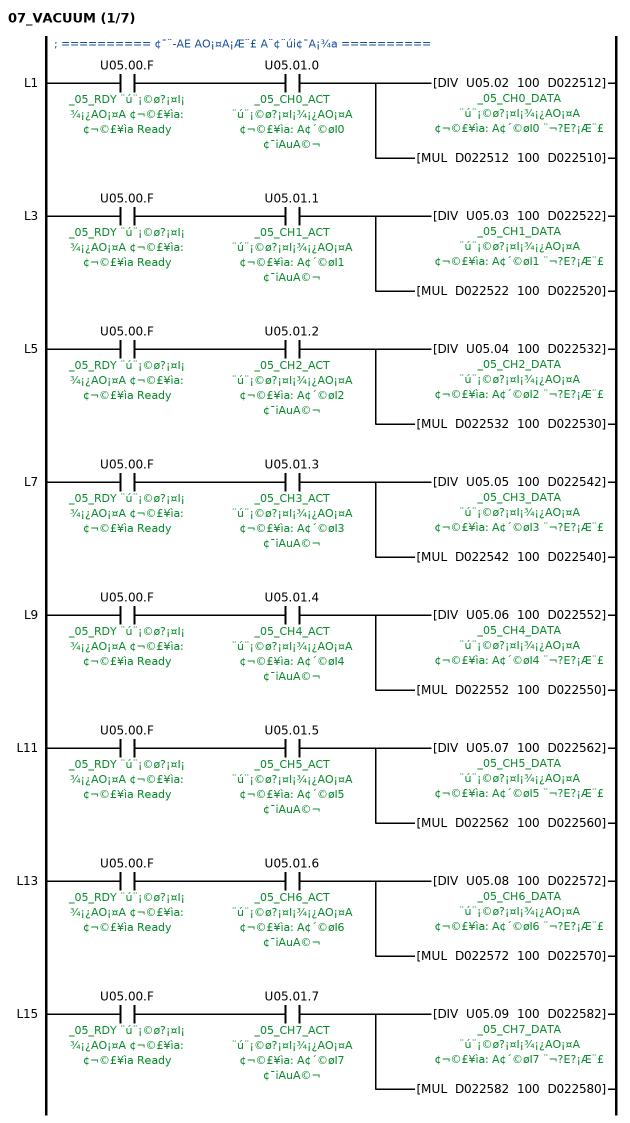
[picture p48: 07_VACUUM rungs L1-L15]
// ========== ¢¯¨­AE AO¡¤A¡Æ¨£ A¨¢¨úi¢¯A¡¾a ==========
; L1
LOAD      U05.00.F	// _05_RDY ¨ú¨¡©ø?¡¤I¡¾¡¿AO¡¤A ¢¬©£¥ìa: ¢¬©£¥ìa Ready
AND       U05.01.0	// _05_CH0_ACT ¨ú¨¡©ø?¡¤I¡¾¡¿AO¡¤A ¢¬©£¥ìa: A¢´©øI0 ¢¯iAuA©¬
DIV       U05.02 100 D022512	// _05_CH0_DATA ¨ú¨¡©ø?¡¤I¡¾¡¿AO¡¤A ¢¬©£¥ìa: A¢´©øI0 ¨¬?E?¡Æ¨£
MUL       D022512 100 D022510
; L3
LOAD      U05.00.F	// _05_RDY ¨ú¨¡©ø?¡¤I¡¾¡¿AO¡¤A ¢¬©£¥ìa: ¢¬©£¥ìa Ready
AND       U05.01.1	// _05_CH1_ACT ¨ú¨¡©ø?¡¤I¡¾¡¿AO¡¤A ¢¬©£¥ìa: A¢´©øI1 ¢¯iAuA©¬
DIV       U05.03 100 D022522	// _05_CH1_DATA ¨ú¨¡©ø?¡¤I¡¾¡¿AO¡¤A ¢¬©£¥ìa: A¢´©øI1 ¨¬?E?¡Æ¨£
MUL       D022522 100 D022520
; L5
LOAD      U05.00.F	// _05_RDY ¨ú¨¡©ø?¡¤I¡¾¡¿AO¡¤A ¢¬©£¥ìa: ¢¬©£¥ìa Ready
AND       U05.01.2	// _05_CH2_ACT ¨ú¨¡©ø?¡¤I¡¾¡¿AO¡¤A ¢¬©£¥ìa: A¢´©øI2 ¢¯iAuA©¬
DIV       U05.04 100 D022532	// _05_CH2_DATA ¨ú¨¡©ø?¡¤I¡¾¡¿AO¡¤A ¢¬©£¥ìa: A¢´©øI2 ¨¬?E?¡Æ¨£
MUL       D022532 100 D022530
; L7
LOAD      U05.00.F	// _05_RDY ¨ú¨¡©ø?¡¤I¡¾¡¿AO¡¤A ¢¬©£¥ìa: ¢¬©£¥ìa Ready
AND       U05.01.3	// _05_CH3_ACT ¨ú¨¡©ø?¡¤I¡¾¡¿AO¡¤A ¢¬©£¥ìa: A¢´©øI3 ¢¯iAuA©¬
DIV       U05.05 100 D022542	// _05_CH3_DATA ¨ú¨¡©ø?¡¤I¡¾¡¿AO¡¤A ¢¬©£¥ìa: A¢´©øI3 ¨¬?E?¡Æ¨£
MUL       D022542 100 D022540
; L9
LOAD      U05.00.F	// _05_RDY ¨ú¨¡©ø?¡¤I¡¾¡¿AO¡¤A ¢¬©£¥ìa: ¢¬©£¥ìa Ready
AND       U05.01.4	// _05_CH4_ACT ¨ú¨¡©ø?¡¤I¡¾¡¿AO¡¤A ¢¬©£¥ìa: A¢´©øI4 ¢¯iAuA©¬
DIV       U05.06 100 D022552	// _05_CH4_DATA ¨ú¨¡©ø?¡¤I¡¾¡¿AO¡¤A ¢¬©£¥ìa: A¢´©øI4 ¨¬?E?¡Æ¨£
MUL       D022552 100 D022550
; L11
LOAD      U05.00.F	// _05_RDY ¨ú¨¡©ø?¡¤I¡¾¡¿AO¡¤A ¢¬©£¥ìa: ¢¬©£¥ìa Ready
AND       U05.01.5	// _05_CH5_ACT ¨ú¨¡©ø?¡¤I¡¾¡¿AO¡¤A ¢¬©£¥ìa: A¢´©øI5 ¢¯iAuA©¬
DIV       U05.07 100 D022562	// _05_CH5_DATA ¨ú¨¡©ø?¡¤I¡¾¡¿AO¡¤A ¢¬©£¥ìa: A¢´©øI5 ¨¬?E?¡Æ¨£
MUL       D022562 100 D022560
; L13
LOAD      U05.00.F	// _05_RDY ¨ú¨¡©ø?¡¤I¡¾¡¿AO¡¤A ¢¬©£¥ìa: ¢¬©£¥ìa Ready
AND       U05.01.6	// _05_CH6_ACT ¨ú¨¡©ø?¡¤I¡¾¡¿AO¡¤A ¢¬©£¥ìa: A¢´©øI6 ¢¯iAuA©¬
DIV       U05.08 100 D022572	// _05_CH6_DATA ¨ú¨¡©ø?¡¤I¡¾¡¿AO¡¤A ¢¬©£¥ìa: A¢´©øI6 ¨¬?E?¡Æ¨£
MUL       D022572 100 D022570
; L15
LOAD      U05.00.F	// _05_RDY ¨ú¨¡©ø?¡¤I¡¾¡¿AO¡¤A ¢¬©£¥ìa: ¢¬©£¥ìa Ready
AND       U05.01.7	// _05_CH7_ACT ¨ú¨¡©ø?¡¤I¡¾¡¿AO¡¤A ¢¬©£¥ìa: A¢´©øI7 ¢¯iAuA©¬
DIV       U05.09 100 D022582	// _05_CH7_DATA ¨ú¨¡©ø?¡¤I¡¾¡¿AO¡¤A ¢¬©£¥ìa: A¢´©øI7 ¨¬?E?¡Æ¨£
MUL       D022582 100 D022580

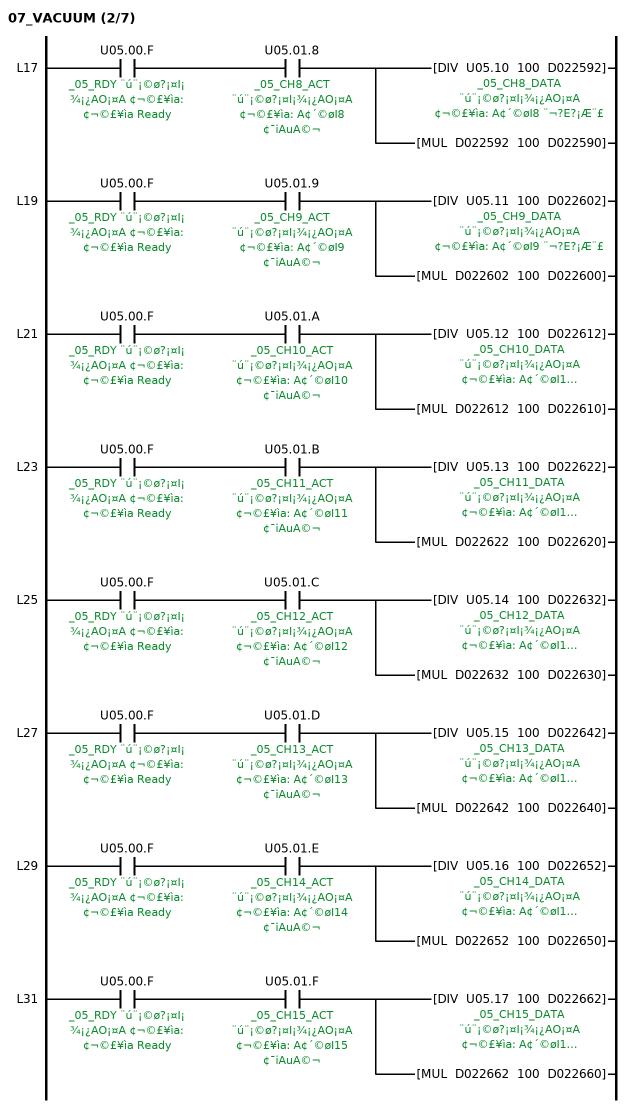
; L17
LOAD      U05.00.F	// _05_RDY ¨ú¨¡©ø?¡¤I¡¾¡¿AO¡¤A ¢¬©£¥ìa: ¢¬©£¥ìa Ready
AND       U05.01.8	// _05_CH8_ACT ¨ú¨¡©ø?¡¤I¡¾¡¿AO¡¤A ¢¬©£¥ìa: A¢´©øI8 ¢¯iAuA©¬
DIV       U05.10 100 D022592	// _05_CH8_DATA ¨ú¨¡©ø?¡¤I¡¾¡¿AO¡¤A ¢¬©£¥ìa: A¢´©øI8 ¨¬?E?¡Æ¨£
MUL       D022592 100 D022590
; L19
LOAD      U05.00.F	// _05_RDY ¨ú¨¡©ø?¡¤I¡¾¡¿AO¡¤A ¢¬©£¥ìa: ¢¬©£¥ìa Ready
AND       U05.01.9	// _05_CH9_ACT ¨ú¨¡©ø?¡¤I¡¾¡¿AO¡¤A ¢¬©£¥ìa: A¢´©øI9 ¢¯iAuA©¬
DIV       U05.11 100 D022602	// _05_CH9_DATA ¨ú¨¡©ø?¡¤I¡¾¡¿AO¡¤A ¢¬©£¥ìa: A¢´©øI9 ¨¬?E?¡Æ¨£
MUL       D022602 100 D022600
; L21
LOAD      U05.00.F	// _05_RDY ¨ú¨¡©ø?¡¤I¡¾¡¿AO¡¤A ¢¬©£¥ìa: ¢¬©£¥ìa Ready
AND       U05.01.A	// _05_CH10_ACT ¨ú¨¡©ø?¡¤I¡¾¡¿AO¡¤A ¢¬©£¥ìa: A¢´©øI10 ¢¯iAuA©¬
DIV       U05.12 100 D022612	// _05_CH10_DATA ¨ú¨¡©ø?¡¤I¡¾¡¿AO¡¤A ¢¬©£¥ìa: A¢´©øI10 ¨¬?E?¡Æ¨£
MUL       D022612 100 D022610
; L23
LOAD      U05.00.F	// _05_RDY ¨ú¨¡©ø?¡¤I¡¾¡¿AO¡¤A ¢¬©£¥ìa: ¢¬©£¥ìa Ready
AND       U05.01.B	// _05_CH11_ACT ¨ú¨¡©ø?¡¤I¡¾¡¿AO¡¤A ¢¬©£¥ìa: A¢´©øI11 ¢¯iAuA©¬
DIV       U05.13 100 D022622	// _05_CH11_DATA ¨ú¨¡©ø?¡¤I¡¾¡¿AO¡¤A ¢¬©£¥ìa: A¢´©øI11 ¨¬?E?¡Æ¨£
MUL       D022622 100 D022620
; L25
LOAD      U05.00.F	// _05_RDY ¨ú¨¡©ø?¡¤I¡¾¡¿AO¡¤A ¢¬©£¥ìa: ¢¬©£¥ìa Ready
AND       U05.01.C	// _05_CH12_ACT ¨ú¨¡©ø?¡¤I¡¾¡¿AO¡¤A ¢¬©£¥ìa: A¢´©øI12 ¢¯iAuA©¬
DIV       U05.14 100 D022632	// _05_CH12_DATA ¨ú¨¡©ø?¡¤I¡¾¡¿AO¡¤A ¢¬©£¥ìa: A¢´©øI12 ¨¬?E?¡Æ¨£
MUL       D022632 100 D022630
; L27
LOAD      U05.00.F	// _05_RDY ¨ú¨¡©ø?¡¤I¡¾¡¿AO¡¤A ¢¬©£¥ìa: ¢¬©£¥ìa Ready
AND       U05.01.D	// _05_CH13_ACT ¨ú¨¡©ø?¡¤I¡¾¡¿AO¡¤A ¢¬©£¥ìa: A¢´©øI13 ¢¯iAuA©¬
DIV       U05.15 100 D022642	// _05_CH13_DATA ¨ú¨¡©ø?¡¤I¡¾¡¿AO¡¤A ¢¬©£¥ìa: A¢´©øI13 ¨¬?E?¡Æ¨£
MUL       D022642 100 D022640
; L29
LOAD      U05.00.F	// _05_RDY ¨ú¨¡©ø?¡¤I¡¾¡¿AO¡¤A ¢¬©£¥ìa: ¢¬©£¥ìa Ready
AND       U05.01.E	// _05_CH14_ACT ¨ú¨¡©ø?¡¤I¡¾¡¿AO¡¤A ¢¬©£¥ìa: A¢´©øI14 ¢¯iAuA©¬
DIV       U05.16 100 D022652	// _05_CH14_DATA ¨ú¨¡©ø?¡¤I¡¾¡¿AO¡¤A ¢¬©£¥ìa: A¢´©øI14 ¨¬?E?¡Æ¨£
MUL       D022652 100 D022650
; L31
LOAD      U05.00.F	// _05_RDY ¨ú¨¡©ø?¡¤I¡¾¡¿AO¡¤A ¢¬©£¥ìa: ¢¬©£¥ìa Ready
AND       U05.01.F	// _05_CH15_ACT ¨ú¨¡©ø?¡¤I¡¾¡¿AO¡¤A ¢¬©£¥ìa: A¢´©øI15 ¢¯iAuA©¬
DIV       U05.17 100 D022662	// _05_CH15_DATA ¨ú¨¡©ø?¡¤I¡¾¡¿AO¡¤A ¢¬©£¥ìa: A¢´©øI15 ¨¬?E?¡Æ¨£
MUL       D022662 100 D022660

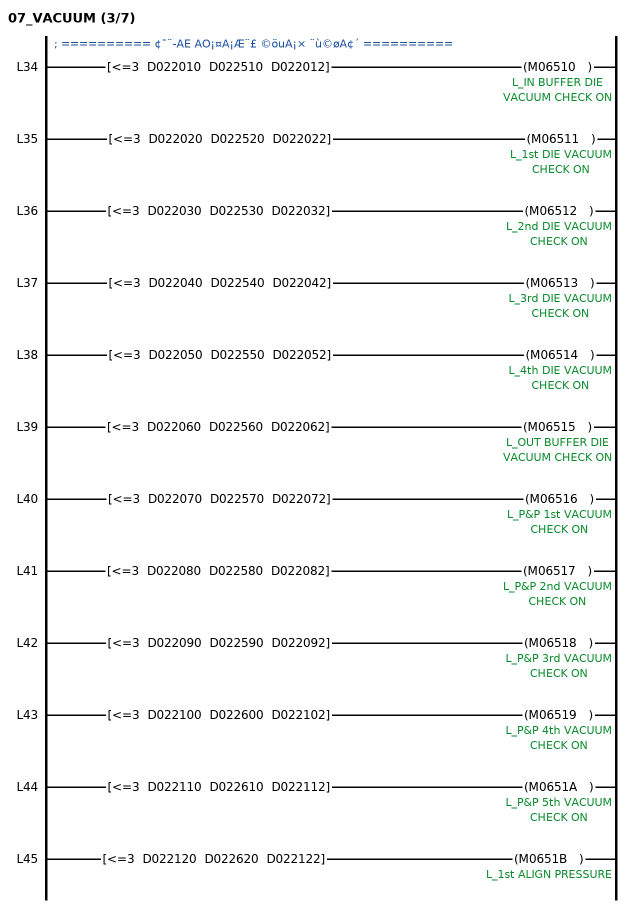
// ========== ¢¯¨­AE AO¡¤A¡Æ¨£ ©öuA¡× ¨ù©øA¢´ ==========
; L34
LOAD<=3   D022010 D022510 D022012
OUT       M06510	// L_IN BUFFER DIE VACUUM CHECK ON
; L35
LOAD<=3   D022020 D022520 D022022
OUT       M06511	// L_1st DIE VACUUM CHECK ON
; L36
LOAD<=3   D022030 D022530 D022032
OUT       M06512	// L_2nd DIE VACUUM CHECK ON
; L37
LOAD<=3   D022040 D022540 D022042
OUT       M06513	// L_3rd DIE VACUUM CHECK ON
; L38
LOAD<=3   D022050 D022550 D022052
OUT       M06514	// L_4th DIE VACUUM CHECK ON
; L39
LOAD<=3   D022060 D022560 D022062
OUT       M06515	// L_OUT BUFFER DIE VACUUM CHECK ON
; L40
LOAD<=3   D022070 D022570 D022072
OUT       M06516	// L_P&P 1st VACUUM CHECK ON
; L41
LOAD<=3   D022080 D022580 D022082
OUT       M06517	// L_P&P 2nd VACUUM CHECK ON
; L42
LOAD<=3   D022090 D022590 D022092
OUT       M06518	// L_P&P 3rd VACUUM CHECK ON
; L43
LOAD<=3   D022100 D022600 D022102
OUT       M06519	// L_P&P 4th VACUUM CHECK ON
; L44
LOAD<=3   D022110 D022610 D022112
OUT       M0651A	// L_P&P 5th VACUUM CHECK ON
; L45
LOAD<=3   D022120 D022620 D022122
OUT       M0651B	// L_1st ALIGN PRESSURE

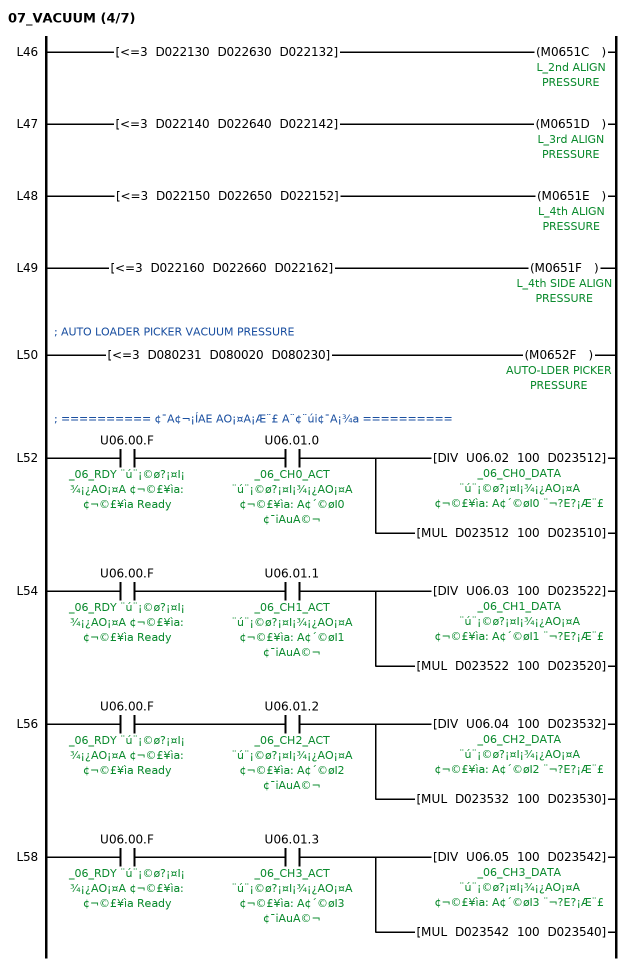
; L46
LOAD<=3   D022130 D022630 D022132
OUT       M0651C	// L_2nd ALIGN PRESSURE
; L47
LOAD<=3   D022140 D022640 D022142
OUT       M0651D	// L_3rd ALIGN PRESSURE
; L48
LOAD<=3   D022150 D022650 D022152
OUT       M0651E	// L_4th ALIGN PRESSURE
; L49
LOAD<=3   D022160 D022660 D022162
OUT       M0651F	// L_4th SIDE ALIGN PRESSURE
; L50
LOAD<=3   D080231 D080020 D080230
OUT       M0652F	// AUTO-LDER PICKER PRESSURE
// output comment: AUTO LOADER PICKER VACUUM PRESSURE
// ========== ¢¯A¢¬¡ÍAE AO¡¤A¡Æ¨£ A¨¢¨úi¢¯A¡¾a ==========
; L52
LOAD      U06.00.F	// _06_RDY ¨ú¨¡©ø?¡¤I¡¾¡¿AO¡¤A ¢¬©£¥ìa: ¢¬©£¥ìa Ready
AND       U06.01.0	// _06_CH0_ACT ¨ú¨¡©ø?¡¤I¡¾¡¿AO¡¤A ¢¬©£¥ìa: A¢´©øI0 ¢¯iAuA©¬
DIV       U06.02 100 D023512	// _06_CH0_DATA ¨ú¨¡©ø?¡¤I¡¾¡¿AO¡¤A ¢¬©£¥ìa: A¢´©øI0 ¨¬?E?¡Æ¨£
MUL       D023512 100 D023510
; L54
LOAD      U06.00.F	// _06_RDY ¨ú¨¡©ø?¡¤I¡¾¡¿AO¡¤A ¢¬©£¥ìa: ¢¬©£¥ìa Ready
AND       U06.01.1	// _06_CH1_ACT ¨ú¨¡©ø?¡¤I¡¾¡¿AO¡¤A ¢¬©£¥ìa: A¢´©øI1 ¢¯iAuA©¬
DIV       U06.03 100 D023522	// _06_CH1_DATA ¨ú¨¡©ø?¡¤I¡¾¡¿AO¡¤A ¢¬©£¥ìa: A¢´©øI1 ¨¬?E?¡Æ¨£
MUL       D023522 100 D023520
; L56
LOAD      U06.00.F	// _06_RDY ¨ú¨¡©ø?¡¤I¡¾¡¿AO¡¤A ¢¬©£¥ìa: ¢¬©£¥ìa Ready
AND       U06.01.2	// _06_CH2_ACT ¨ú¨¡©ø?¡¤I¡¾¡¿AO¡¤A ¢¬©£¥ìa: A¢´©øI2 ¢¯iAuA©¬
DIV       U06.04 100 D023532	// _06_CH2_DATA ¨ú¨¡©ø?¡¤I¡¾¡¿AO¡¤A ¢¬©£¥ìa: A¢´©øI2 ¨¬?E?¡Æ¨£
MUL       D023532 100 D023530
; L58
LOAD      U06.00.F	// _06_RDY ¨ú¨¡©ø?¡¤I¡¾¡¿AO¡¤A ¢¬©£¥ìa: ¢¬©£¥ìa Ready
AND       U06.01.3	// _06_CH3_ACT ¨ú¨¡©ø?¡¤I¡¾¡¿AO¡¤A ¢¬©£¥ìa: A¢´©øI3 ¢¯iAuA©¬
DIV       U06.05 100 D023542	// _06_CH3_DATA ¨ú¨¡©ø?¡¤I¡¾¡¿AO¡¤A ¢¬©£¥ìa: A¢´©øI3 ¨¬?E?¡Æ¨£
MUL       D023542 100 D023540

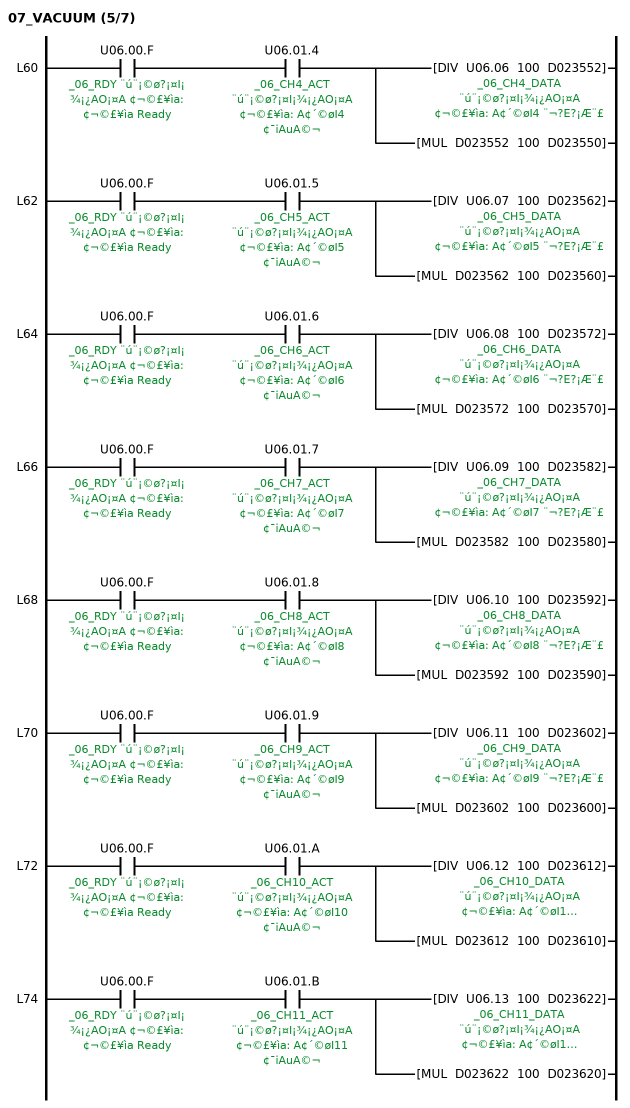
; L60
LOAD      U06.00.F	// _06_RDY ¨ú¨¡©ø?¡¤I¡¾¡¿AO¡¤A ¢¬©£¥ìa: ¢¬©£¥ìa Ready
AND       U06.01.4	// _06_CH4_ACT ¨ú¨¡©ø?¡¤I¡¾¡¿AO¡¤A ¢¬©£¥ìa: A¢´©øI4 ¢¯iAuA©¬
DIV       U06.06 100 D023552	// _06_CH4_DATA ¨ú¨¡©ø?¡¤I¡¾¡¿AO¡¤A ¢¬©£¥ìa: A¢´©øI4 ¨¬?E?¡Æ¨£
MUL       D023552 100 D023550
; L62
LOAD      U06.00.F	// _06_RDY ¨ú¨¡©ø?¡¤I¡¾¡¿AO¡¤A ¢¬©£¥ìa: ¢¬©£¥ìa Ready
AND       U06.01.5	// _06_CH5_ACT ¨ú¨¡©ø?¡¤I¡¾¡¿AO¡¤A ¢¬©£¥ìa: A¢´©øI5 ¢¯iAuA©¬
DIV       U06.07 100 D023562	// _06_CH5_DATA ¨ú¨¡©ø?¡¤I¡¾¡¿AO¡¤A ¢¬©£¥ìa: A¢´©øI5 ¨¬?E?¡Æ¨£
MUL       D023562 100 D023560
; L64
LOAD      U06.00.F	// _06_RDY ¨ú¨¡©ø?¡¤I¡¾¡¿AO¡¤A ¢¬©£¥ìa: ¢¬©£¥ìa Ready
AND       U06.01.6	// _06_CH6_ACT ¨ú¨¡©ø?¡¤I¡¾¡¿AO¡¤A ¢¬©£¥ìa: A¢´©øI6 ¢¯iAuA©¬
DIV       U06.08 100 D023572	// _06_CH6_DATA ¨ú¨¡©ø?¡¤I¡¾¡¿AO¡¤A ¢¬©£¥ìa: A¢´©øI6 ¨¬?E?¡Æ¨£
MUL       D023572 100 D023570
; L66
LOAD      U06.00.F	// _06_RDY ¨ú¨¡©ø?¡¤I¡¾¡¿AO¡¤A ¢¬©£¥ìa: ¢¬©£¥ìa Ready
AND       U06.01.7	// _06_CH7_ACT ¨ú¨¡©ø?¡¤I¡¾¡¿AO¡¤A ¢¬©£¥ìa: A¢´©øI7 ¢¯iAuA©¬
DIV       U06.09 100 D023582	// _06_CH7_DATA ¨ú¨¡©ø?¡¤I¡¾¡¿AO¡¤A ¢¬©£¥ìa: A¢´©øI7 ¨¬?E?¡Æ¨£
MUL       D023582 100 D023580
; L68
LOAD      U06.00.F	// _06_RDY ¨ú¨¡©ø?¡¤I¡¾¡¿AO¡¤A ¢¬©£¥ìa: ¢¬©£¥ìa Ready
AND       U06.01.8	// _06_CH8_ACT ¨ú¨¡©ø?¡¤I¡¾¡¿AO¡¤A ¢¬©£¥ìa: A¢´©øI8 ¢¯iAuA©¬
DIV       U06.10 100 D023592	// _06_CH8_DATA ¨ú¨¡©ø?¡¤I¡¾¡¿AO¡¤A ¢¬©£¥ìa: A¢´©øI8 ¨¬?E?¡Æ¨£
MUL       D023592 100 D023590
; L70
LOAD      U06.00.F	// _06_RDY ¨ú¨¡©ø?¡¤I¡¾¡¿AO¡¤A ¢¬©£¥ìa: ¢¬©£¥ìa Ready
AND       U06.01.9	// _06_CH9_ACT ¨ú¨¡©ø?¡¤I¡¾¡¿AO¡¤A ¢¬©£¥ìa: A¢´©øI9 ¢¯iAuA©¬
DIV       U06.11 100 D023602	// _06_CH9_DATA ¨ú¨¡©ø?¡¤I¡¾¡¿AO¡¤A ¢¬©£¥ìa: A¢´©øI9 ¨¬?E?¡Æ¨£
MUL       D023602 100 D023600
; L72
LOAD      U06.00.F	// _06_RDY ¨ú¨¡©ø?¡¤I¡¾¡¿AO¡¤A ¢¬©£¥ìa: ¢¬©£¥ìa Ready
AND       U06.01.A	// _06_CH10_ACT ¨ú¨¡©ø?¡¤I¡¾¡¿AO¡¤A ¢¬©£¥ìa: A¢´©øI10 ¢¯iAuA©¬
DIV       U06.12 100 D023612	// _06_CH10_DATA ¨ú¨¡©ø?¡¤I¡¾¡¿AO¡¤A ¢¬©£¥ìa: A¢´©øI10 ¨¬?E?¡Æ¨£
MUL       D023612 100 D023610
; L74
LOAD      U06.00.F	// _06_RDY ¨ú¨¡©ø?¡¤I¡¾¡¿AO¡¤A ¢¬©£¥ìa: ¢¬©£¥ìa Ready
AND       U06.01.B	// _06_CH11_ACT ¨ú¨¡©ø?¡¤I¡¾¡¿AO¡¤A ¢¬©£¥ìa: A¢´©øI11 ¢¯iAuA©¬
DIV       U06.13 100 D023622	// _06_CH11_DATA ¨ú¨¡©ø?¡¤I¡¾¡¿AO¡¤A ¢¬©£¥ìa: A¢´©øI11 ¨¬?E?¡Æ¨£
MUL       D023622 100 D023620

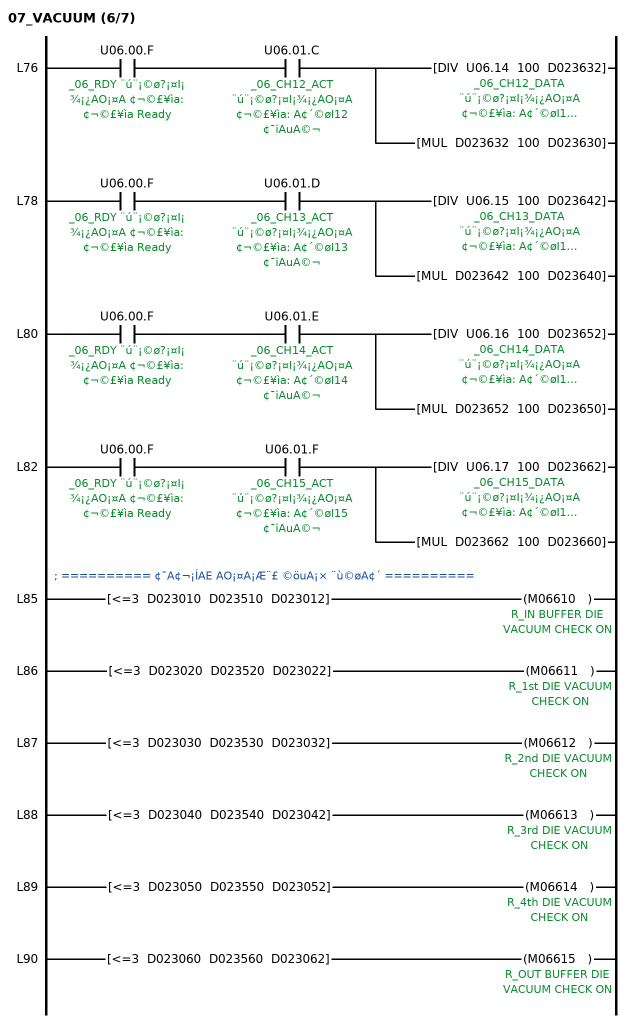
; L76
LOAD      U06.00.F	// _06_RDY ¨ú¨¡©ø?¡¤I¡¾¡¿AO¡¤A ¢¬©£¥ìa: ¢¬©£¥ìa Ready
AND       U06.01.C	// _06_CH12_ACT ¨ú¨¡©ø?¡¤I¡¾¡¿AO¡¤A ¢¬©£¥ìa: A¢´©øI12 ¢¯iAuA©¬
DIV       U06.14 100 D023632	// _06_CH12_DATA ¨ú¨¡©ø?¡¤I¡¾¡¿AO¡¤A ¢¬©£¥ìa: A¢´©øI12 ¨¬?E?¡Æ¨£
MUL       D023632 100 D023630
; L78
LOAD      U06.00.F	// _06_RDY ¨ú¨¡©ø?¡¤I¡¾¡¿AO¡¤A ¢¬©£¥ìa: ¢¬©£¥ìa Ready
AND       U06.01.D	// _06_CH13_ACT ¨ú¨¡©ø?¡¤I¡¾¡¿AO¡¤A ¢¬©£¥ìa: A¢´©øI13 ¢¯iAuA©¬
DIV       U06.15 100 D023642	// _06_CH13_DATA ¨ú¨¡©ø?¡¤I¡¾¡¿AO¡¤A ¢¬©£¥ìa: A¢´©øI13 ¨¬?E?¡Æ¨£
MUL       D023642 100 D023640
; L80
LOAD      U06.00.F	// _06_RDY ¨ú¨¡©ø?¡¤I¡¾¡¿AO¡¤A ¢¬©£¥ìa: ¢¬©£¥ìa Ready
AND       U06.01.E	// _06_CH14_ACT ¨ú¨¡©ø?¡¤I¡¾¡¿AO¡¤A ¢¬©£¥ìa: A¢´©øI14 ¢¯iAuA©¬
DIV       U06.16 100 D023652	// _06_CH14_DATA ¨ú¨¡©ø?¡¤I¡¾¡¿AO¡¤A ¢¬©£¥ìa: A¢´©øI14 ¨¬?E?¡Æ¨£
MUL       D023652 100 D023650
; L82
LOAD      U06.00.F	// _06_RDY ¨ú¨¡©ø?¡¤I¡¾¡¿AO¡¤A ¢¬©£¥ìa: ¢¬©£¥ìa Ready
AND       U06.01.F	// _06_CH15_ACT ¨ú¨¡©ø?¡¤I¡¾¡¿AO¡¤A ¢¬©£¥ìa: A¢´©øI15 ¢¯iAuA©¬
DIV       U06.17 100 D023662	// _06_CH15_DATA ¨ú¨¡©ø?¡¤I¡¾¡¿AO¡¤A ¢¬©£¥ìa: A¢´©øI15 ¨¬?E?¡Æ¨£
MUL       D023662 100 D023660
// ========== ¢¯A¢¬¡ÍAE AO¡¤A¡Æ¨£ ©öuA¡× ¨ù©øA¢´ ==========
; L85
LOAD<=3   D023010 D023510 D023012
OUT       M06610	// R_IN BUFFER DIE VACUUM CHECK ON
; L86
LOAD<=3   D023020 D023520 D023022
OUT       M06611	// R_1st DIE VACUUM CHECK ON
; L87
LOAD<=3   D023030 D023530 D023032
OUT       M06612	// R_2nd DIE VACUUM CHECK ON
; L88
LOAD<=3   D023040 D023540 D023042
OUT       M06613	// R_3rd DIE VACUUM CHECK ON
; L89
LOAD<=3   D023050 D023550 D023052
OUT       M06614	// R_4th DIE VACUUM CHECK ON
; L90
LOAD<=3   D023060 D023560 D023062
OUT       M06615	// R_OUT BUFFER DIE VACUUM CHECK ON

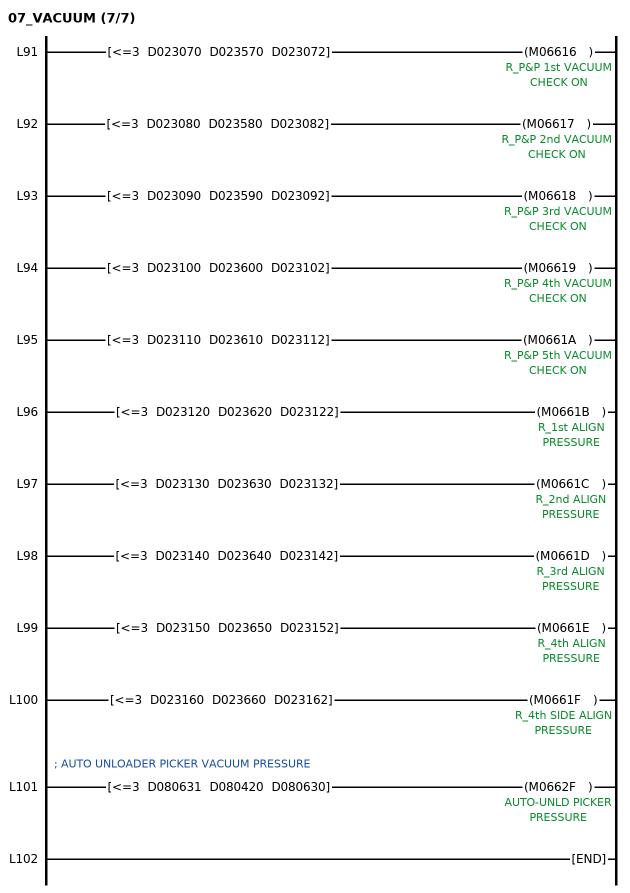
; L91
LOAD<=3   D023070 D023570 D023072
OUT       M06616	// R_P&P 1st VACUUM CHECK ON
; L92
LOAD<=3   D023080 D023580 D023082
OUT       M06617	// R_P&P 2nd VACUUM CHECK ON
; L93
LOAD<=3   D023090 D023590 D023092
OUT       M06618	// R_P&P 3rd VACUUM CHECK ON
; L94
LOAD<=3   D023100 D023600 D023102
OUT       M06619	// R_P&P 4th VACUUM CHECK ON
; L95
LOAD<=3   D023110 D023610 D023112
OUT       M0661A	// R_P&P 5th VACUUM CHECK ON
; L96
LOAD<=3   D023120 D023620 D023122
OUT       M0661B	// R_1st ALIGN PRESSURE
; L97
LOAD<=3   D023130 D023630 D023132
OUT       M0661C	// R_2nd ALIGN PRESSURE
; L98
LOAD<=3   D023140 D023640 D023142
OUT       M0661D	// R_3rd ALIGN PRESSURE
; L99
LOAD<=3   D023150 D023650 D023152
OUT       M0661E	// R_4th ALIGN PRESSURE
; L100
LOAD<=3   D023160 D023660 D023162
OUT       M0661F	// R_4th SIDE ALIGN PRESSURE
; L101
LOAD<=3   D080631 D080420 D080630
OUT       M0662F	// AUTO-UNLD PICKER PRESSURE
// output comment: AUTO UNLOADER PICKER VACUUM PRESSURE
; L102
END

PROGRAM 11_L_1st_MAND (task: ¨ö¨¬A¥ì CA¡¤I¡¾¡¿¡¤¡Í)

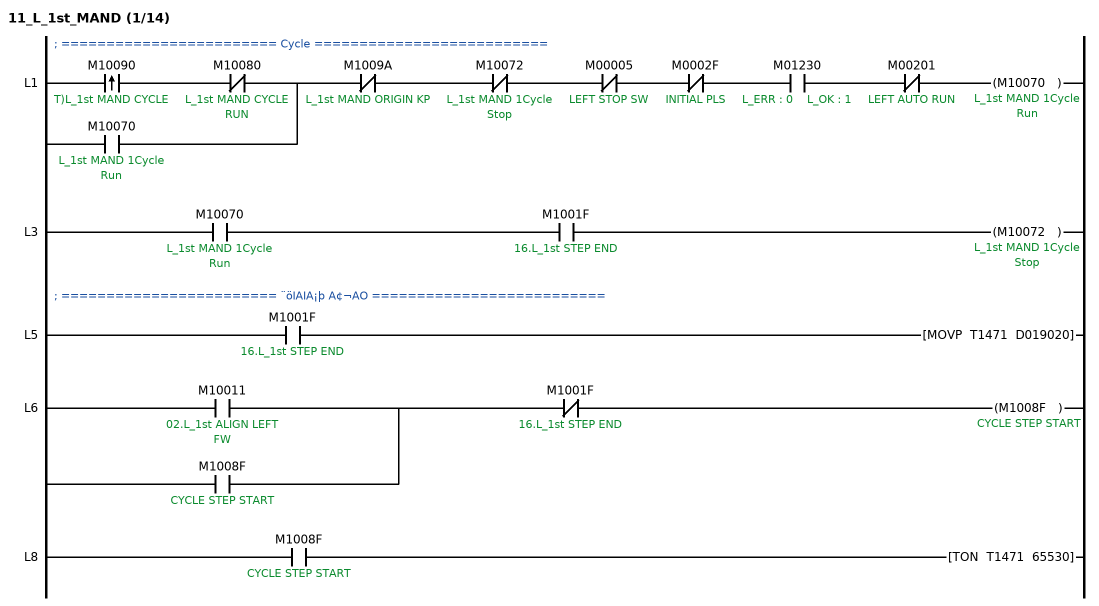
// ======================== Cycle ==========================
; L1
LOADP     M10090	// T)L_1st MAND CYCLE
AND NOT   M10080	// L_1st MAND CYCLE RUN
OR        M10070	// L_1st MAND 1Cycle Run
AND NOT   M1009A	// L_1st MAND ORIGIN KP
AND NOT   M10072	// L_1st MAND 1Cycle Stop
AND NOT   M00005	// LEFT STOP SW
AND NOT   M0002F	// INITIAL PLS
AND       M01230	// L_ERR : 0    L_OK : 1
AND NOT   M00201	// LEFT AUTO RUN
OUT       M10070	// L_1st MAND 1Cycle Run
; L3
LOAD      M10070	// L_1st MAND 1Cycle Run
AND       M1001F	// 16.L_1st STEP END
OUT       M10072	// L_1st MAND 1Cycle Stop
// ======================== ¨öIAIA¡þ A¢¬AO ==========================
; L5
LOAD      M1001F	// 16.L_1st STEP END
MOVP      T1471 D019020
; L6
LOAD      M10011	// 02.L_1st ALIGN LEFT FW
OR        M1008F	// CYCLE STEP START
AND NOT   M1001F	// 16.L_1st STEP END
OUT       M1008F	// CYCLE STEP START
; L8
LOAD      M1008F	// CYCLE STEP START
TON       T1471 65530

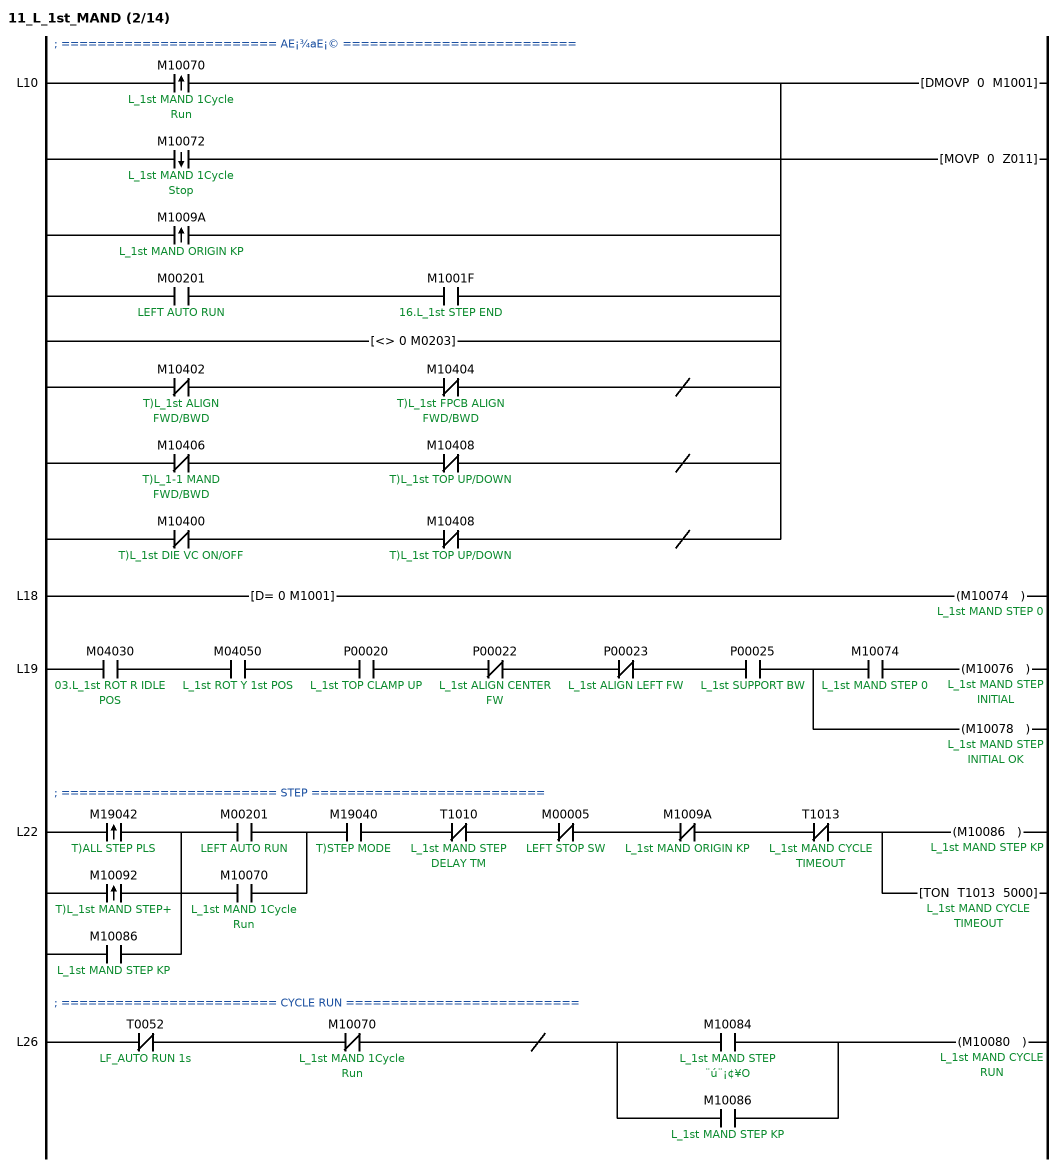
// ======================== AE¡¾aE¡© ==========================
; L10
LOADP     M10070	// L_1st MAND 1Cycle Run
ORN       M10072	// L_1st MAND 1Cycle Stop
ORP       M1009A	// L_1st MAND ORIGIN KP
LOAD      M00201	// LEFT AUTO RUN
AND       M1001F	// 16.L_1st STEP END
OR LOAD
OR<>      0 M0203
LOAD NOT  M10402	// T)L_1st ALIGN FWD/BWD
AND NOT   M10404	// T)L_1st FPCB ALIGN FWD/BWD
NOT
OR LOAD
LOAD NOT  M10406	// T)L_1-1 MAND FWD/BWD
AND NOT   M10408	// T)L_1st TOP UP/DOWN
NOT
OR LOAD
LOAD NOT  M10400	// T)L_1st DIE VC ON/OFF
AND NOT   M10408	// T)L_1st TOP UP/DOWN
NOT
OR LOAD
DMOVP     0 M1001
MOVP      0 Z011
; L18
LOADD=    0 M1001
OUT       M10074	// L_1st MAND STEP 0
; L19
LOAD      M04030	// 03.L_1st ROT R IDLE POS
AND       M04050	// L_1st ROT Y 1st POS
AND       P00020	// L_1st TOP CLAMP UP
AND NOT   P00022	// L_1st ALIGN CENTER FW
AND NOT   P00023	// L_1st ALIGN LEFT FW
AND       P00025	// L_1st SUPPORT BW
MPUSH
AND       M10074	// L_1st MAND STEP 0
OUT       M10076	// L_1st MAND STEP INITIAL
MPOP
OUT       M10078	// L_1st MAND STEP INITIAL OK
// ======================== STEP ==========================
; L22
LOADP     M19042	// T)ALL STEP PLS
ORP       M10092	// T)L_1st MAND STEP+
OR        M10086	// L_1st MAND STEP KP
LOAD      M00201	// LEFT AUTO RUN
OR        M10070	// L_1st MAND 1Cycle Run
AND LOAD
AND       M19040	// T)STEP MODE
AND NOT   T1010	// L_1st MAND STEP DELAY TM
AND NOT   M00005	// LEFT STOP SW
AND NOT   M1009A	// L_1st MAND ORIGIN KP
AND NOT   T1013	// L_1st MAND CYCLE TIMEOUT
OUT       M10086	// L_1st MAND STEP KP
TON       T1013 5000	// L_1st MAND CYCLE TIMEOUT
// ======================== CYCLE RUN ==========================
; L26
LOAD NOT  T0052	// LF_AUTO RUN 1s
AND NOT   M10070	// L_1st MAND 1Cycle Run
NOT
LOAD      M10084	// L_1st MAND STEP ¨ú¨¡¢¥O
OR        M10086	// L_1st MAND STEP KP
AND LOAD
OUT       M10080	// L_1st MAND CYCLE RUN

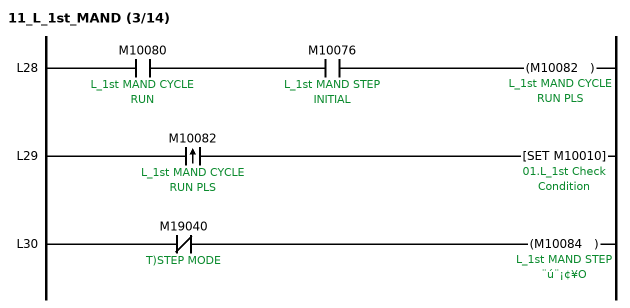
; L28
LOAD      M10080	// L_1st MAND CYCLE RUN
AND       M10076	// L_1st MAND STEP INITIAL
OUT       M10082	// L_1st MAND CYCLE RUN PLS
; L29
LOADP     M10082	// L_1st MAND CYCLE RUN PLS
SET       M10010	// 01.L_1st Check Condition
; L30
LOAD NOT  M19040	// T)STEP MODE
OUT       M10084	// L_1st MAND STEP ¨ú¨¡¢¥O

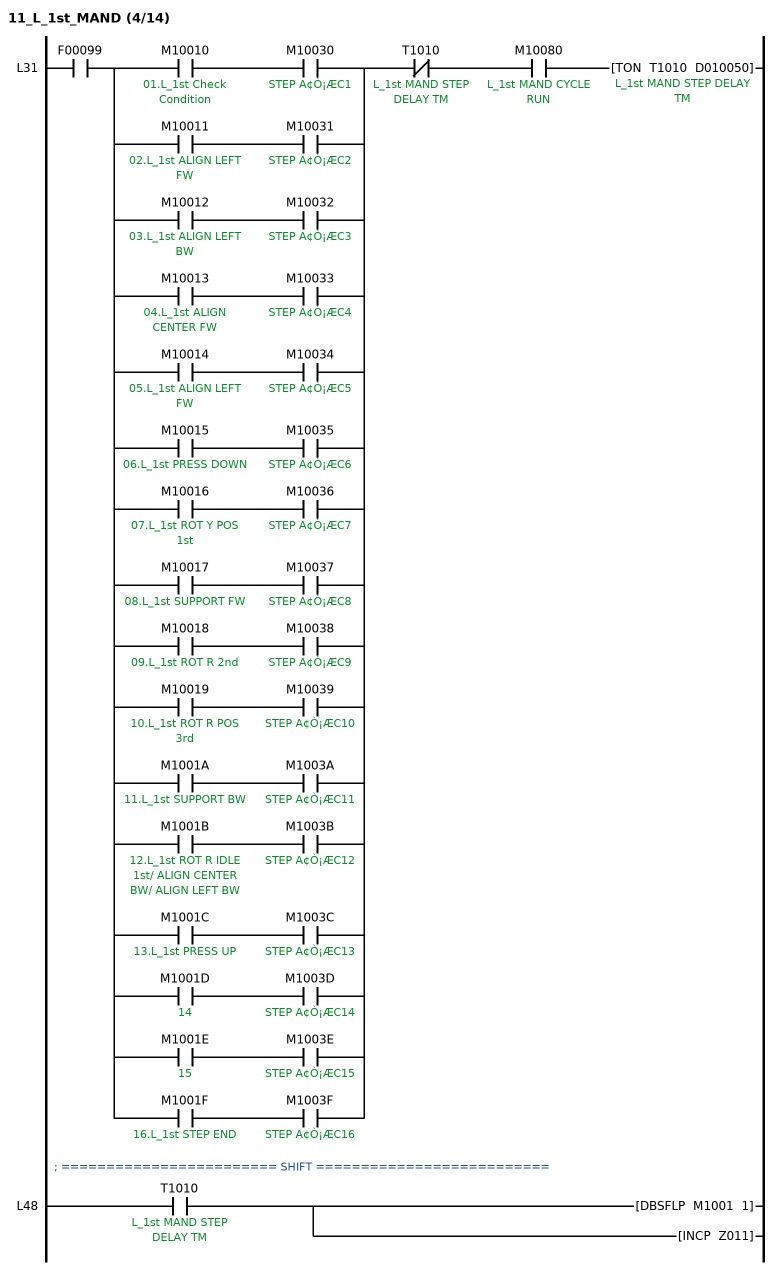
; L31
LOAD      F00099
LOAD      M10010	// 01.L_1st Check Condition
AND       M10030	// STEP A¢Ò¡ÆC1
LOAD      M10011	// 02.L_1st ALIGN LEFT FW
AND       M10031	// STEP A¢Ò¡ÆC2
OR LOAD
LOAD      M10012	// 03.L_1st ALIGN LEFT BW
AND       M10032	// STEP A¢Ò¡ÆC3
OR LOAD
LOAD      M10013	// 04.L_1st ALIGN CENTER FW
AND       M10033	// STEP A¢Ò¡ÆC4
OR LOAD
LOAD      M10014	// 05.L_1st ALIGN LEFT FW
AND       M10034	// STEP A¢Ò¡ÆC5
OR LOAD
LOAD      M10015	// 06.L_1st PRESS DOWN
AND       M10035	// STEP A¢Ò¡ÆC6
OR LOAD
LOAD      M10016	// 07.L_1st ROT Y POS 1st
AND       M10036	// STEP A¢Ò¡ÆC7
OR LOAD
LOAD      M10017	// 08.L_1st SUPPORT FW
AND       M10037	// STEP A¢Ò¡ÆC8
OR LOAD
LOAD      M10018	// 09.L_1st ROT R 2nd
AND       M10038	// STEP A¢Ò¡ÆC9
OR LOAD
LOAD      M10019	// 10.L_1st ROT R POS 3rd
AND       M10039	// STEP A¢Ò¡ÆC10
OR LOAD
LOAD      M1001A	// 11.L_1st SUPPORT BW
AND       M1003A	// STEP A¢Ò¡ÆC11
OR LOAD
LOAD      M1001B	// 12.L_1st ROT R IDLE 1st/ ALIGN CENTER BW/ ALIGN LEFT BW
AND       M1003B	// STEP A¢Ò¡ÆC12
OR LOAD
LOAD      M1001C	// 13.L_1st PRESS UP
AND       M1003C	// STEP A¢Ò¡ÆC13
OR LOAD
LOAD      M1001D	// 14
AND       M1003D	// STEP A¢Ò¡ÆC14
OR LOAD
LOAD      M1001E	// 15
AND       M1003E	// STEP A¢Ò¡ÆC15
OR LOAD
LOAD      M1001F	// 16.L_1st STEP END
AND       M1003F	// STEP A¢Ò¡ÆC16
OR LOAD
AND LOAD
AND NOT   T1010	// L_1st MAND STEP DELAY TM
AND       M10080	// L_1st MAND CYCLE RUN
TON       T1010 D010050	// L_1st MAND STEP DELAY TM
// ======================== SHIFT ==========================
; L48
LOAD      T1010	// L_1st MAND STEP DELAY TM
DBSFLP    M1001 1
INCP      Z011

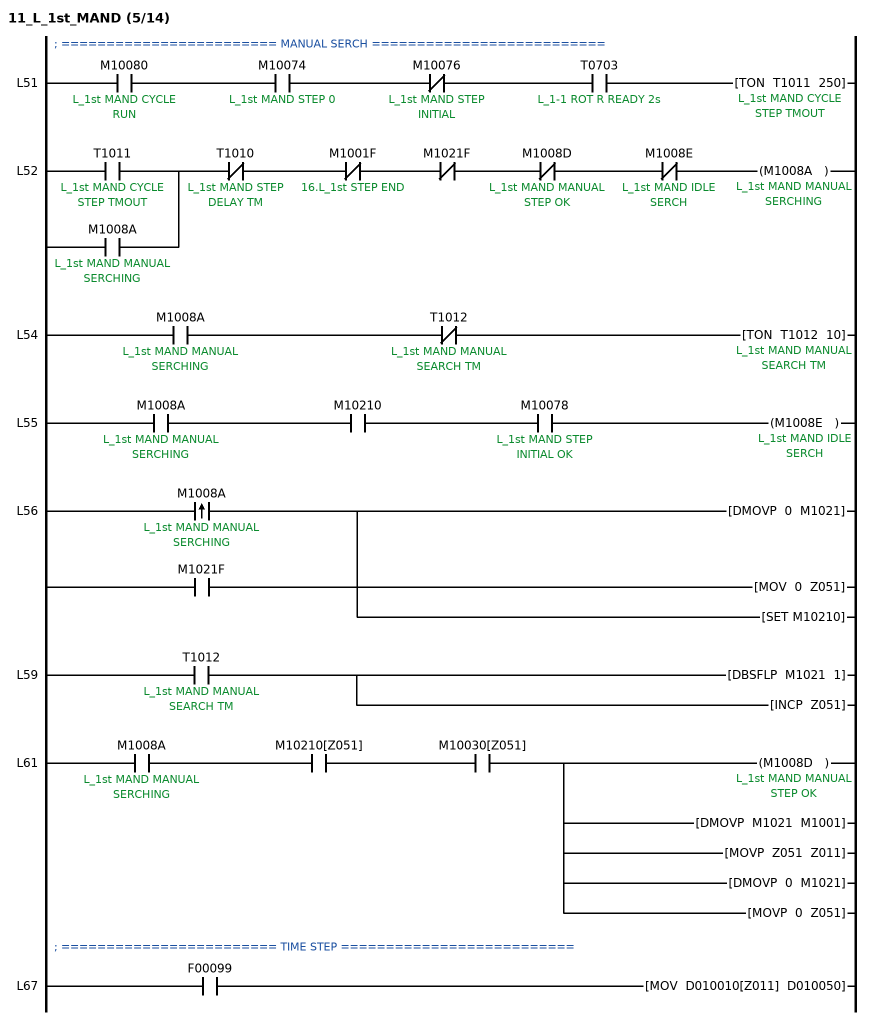
// ======================== MANUAL SERCH ==========================
; L51
LOAD      M10080	// L_1st MAND CYCLE RUN
AND       M10074	// L_1st MAND STEP 0
AND NOT   M10076	// L_1st MAND STEP INITIAL
AND       T0703	// L_1-1 ROT R READY 2s
TON       T1011 250	// L_1st MAND CYCLE STEP TMOUT
; L52
LOAD      T1011	// L_1st MAND CYCLE STEP TMOUT
OR        M1008A	// L_1st MAND MANUAL SERCHING
AND NOT   T1010	// L_1st MAND STEP DELAY TM
AND NOT   M1001F	// 16.L_1st STEP END
AND NOT   M1021F
AND NOT   M1008D	// L_1st MAND MANUAL STEP OK
AND NOT   M1008E	// L_1st MAND IDLE SERCH
OUT       M1008A	// L_1st MAND MANUAL SERCHING
; L54
LOAD      M1008A	// L_1st MAND MANUAL SERCHING
AND NOT   T1012	// L_1st MAND MANUAL SEARCH TM
TON       T1012 10	// L_1st MAND MANUAL SEARCH TM
; L55
LOAD      M1008A	// L_1st MAND MANUAL SERCHING
AND       M10210
AND       M10078	// L_1st MAND STEP INITIAL OK
OUT       M1008E	// L_1st MAND IDLE SERCH
; L56
LOADP     M1008A	// L_1st MAND MANUAL SERCHING
OR        M1021F
DMOVP     0 M1021
MOV       0 Z051
SET       M10210
; L59
LOAD      T1012	// L_1st MAND MANUAL SEARCH TM
DBSFLP    M1021 1
INCP      Z051
; L61
LOAD      M1008A	// L_1st MAND MANUAL SERCHING
AND       M10210[Z051]
AND       M10030[Z051]
OUT       M1008D	// L_1st MAND MANUAL STEP OK
DMOVP     M1021 M1001
MOVP      Z051 Z011
DMOVP     0 M1021
MOVP      0 Z051
// ======================== TIME STEP ==========================
; L67
LOAD      F00099
MOV       D010010[Z011] D010050

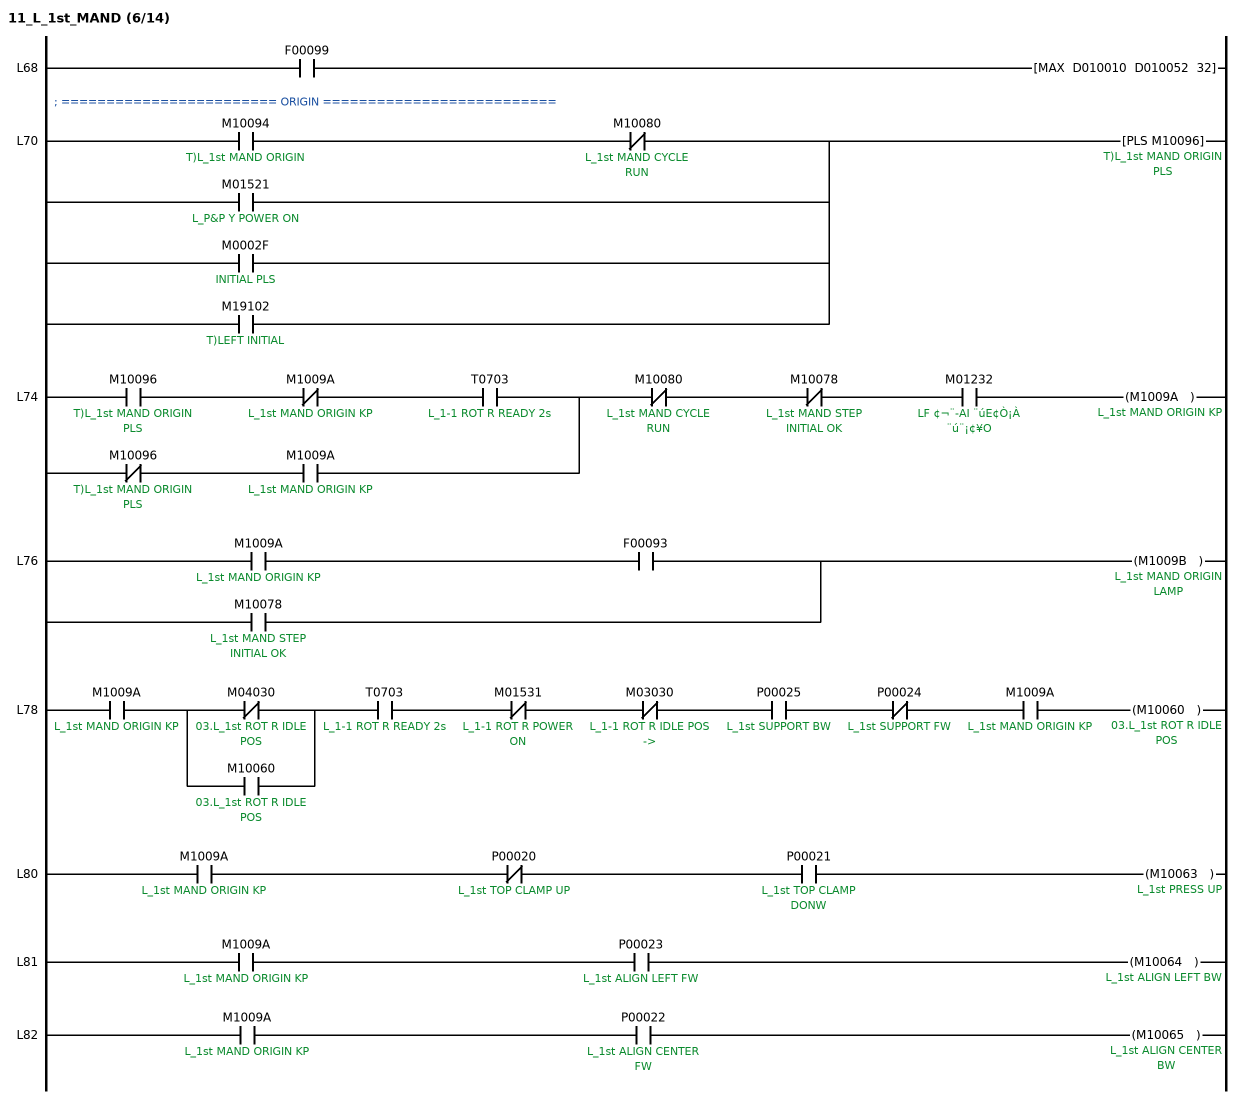
; L68
LOAD      F00099
MAX       D010010 D010052 32
// ======================== ORIGIN ==========================
; L70
LOAD      M10094	// T)L_1st MAND ORIGIN
AND NOT   M10080	// L_1st MAND CYCLE RUN
OR        M01521	// L_P&P Y POWER ON
OR        M0002F	// INITIAL PLS
OR        M19102	// T)LEFT INITIAL
OUTP      M10096	// T)L_1st MAND ORIGIN PLS
; L74
LOAD      M10096	// T)L_1st MAND ORIGIN PLS
AND NOT   M1009A	// L_1st MAND ORIGIN KP
AND       T0703	// L_1-1 ROT R READY 2s
LOAD NOT  M10096	// T)L_1st MAND ORIGIN PLS
AND       M1009A	// L_1st MAND ORIGIN KP
OR LOAD
AND NOT   M10080	// L_1st MAND CYCLE RUN
AND NOT   M10078	// L_1st MAND STEP INITIAL OK
AND       M01232	// LF ¢¬¨­AI ¨úE¢Ò¡À ¨ú¨¡¢¥O
OUT       M1009A	// L_1st MAND ORIGIN KP
; L76
LOAD      M1009A	// L_1st MAND ORIGIN KP
AND       F00093
OR        M10078	// L_1st MAND STEP INITIAL OK
OUT       M1009B	// L_1st MAND ORIGIN LAMP
; L78
LOAD      M1009A	// L_1st MAND ORIGIN KP
LOAD NOT  M04030	// 03.L_1st ROT R IDLE POS
OR        M10060	// 03.L_1st ROT R IDLE POS
AND LOAD
AND       T0703	// L_1-1 ROT R READY 2s
AND NOT   M01531	// L_1-1 ROT R POWER ON
AND NOT   M03030	// L_1-1 ROT R IDLE POS ->
AND       P00025	// L_1st SUPPORT BW
AND NOT   P00024	// L_1st SUPPORT FW
AND       M1009A	// L_1st MAND ORIGIN KP
OUT       M10060	// 03.L_1st ROT R IDLE POS
; L80
LOAD      M1009A	// L_1st MAND ORIGIN KP
AND NOT   P00020	// L_1st TOP CLAMP UP
AND       P00021	// L_1st TOP CLAMP DONW
OUT       M10063	// L_1st PRESS UP
; L81
LOAD      M1009A	// L_1st MAND ORIGIN KP
AND       P00023	// L_1st ALIGN LEFT FW
OUT       M10064	// L_1st ALIGN LEFT BW
; L82
LOAD      M1009A	// L_1st MAND ORIGIN KP
AND       P00022	// L_1st ALIGN CENTER FW
OUT       M10065	// L_1st ALIGN CENTER BW

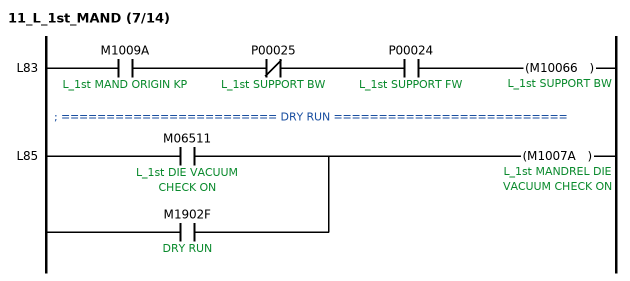
; L83
LOAD      M1009A	// L_1st MAND ORIGIN KP
AND NOT   P00025	// L_1st SUPPORT BW
AND       P00024	// L_1st SUPPORT FW
OUT       M10066	// L_1st SUPPORT BW
// ======================== DRY RUN ==========================
; L85
LOAD      M06511	// L_1st DIE VACUUM CHECK ON
OR        M1902F	// DRY RUN
OUT       M1007A	// L_1st MANDREL DIE VACUUM CHECK ON

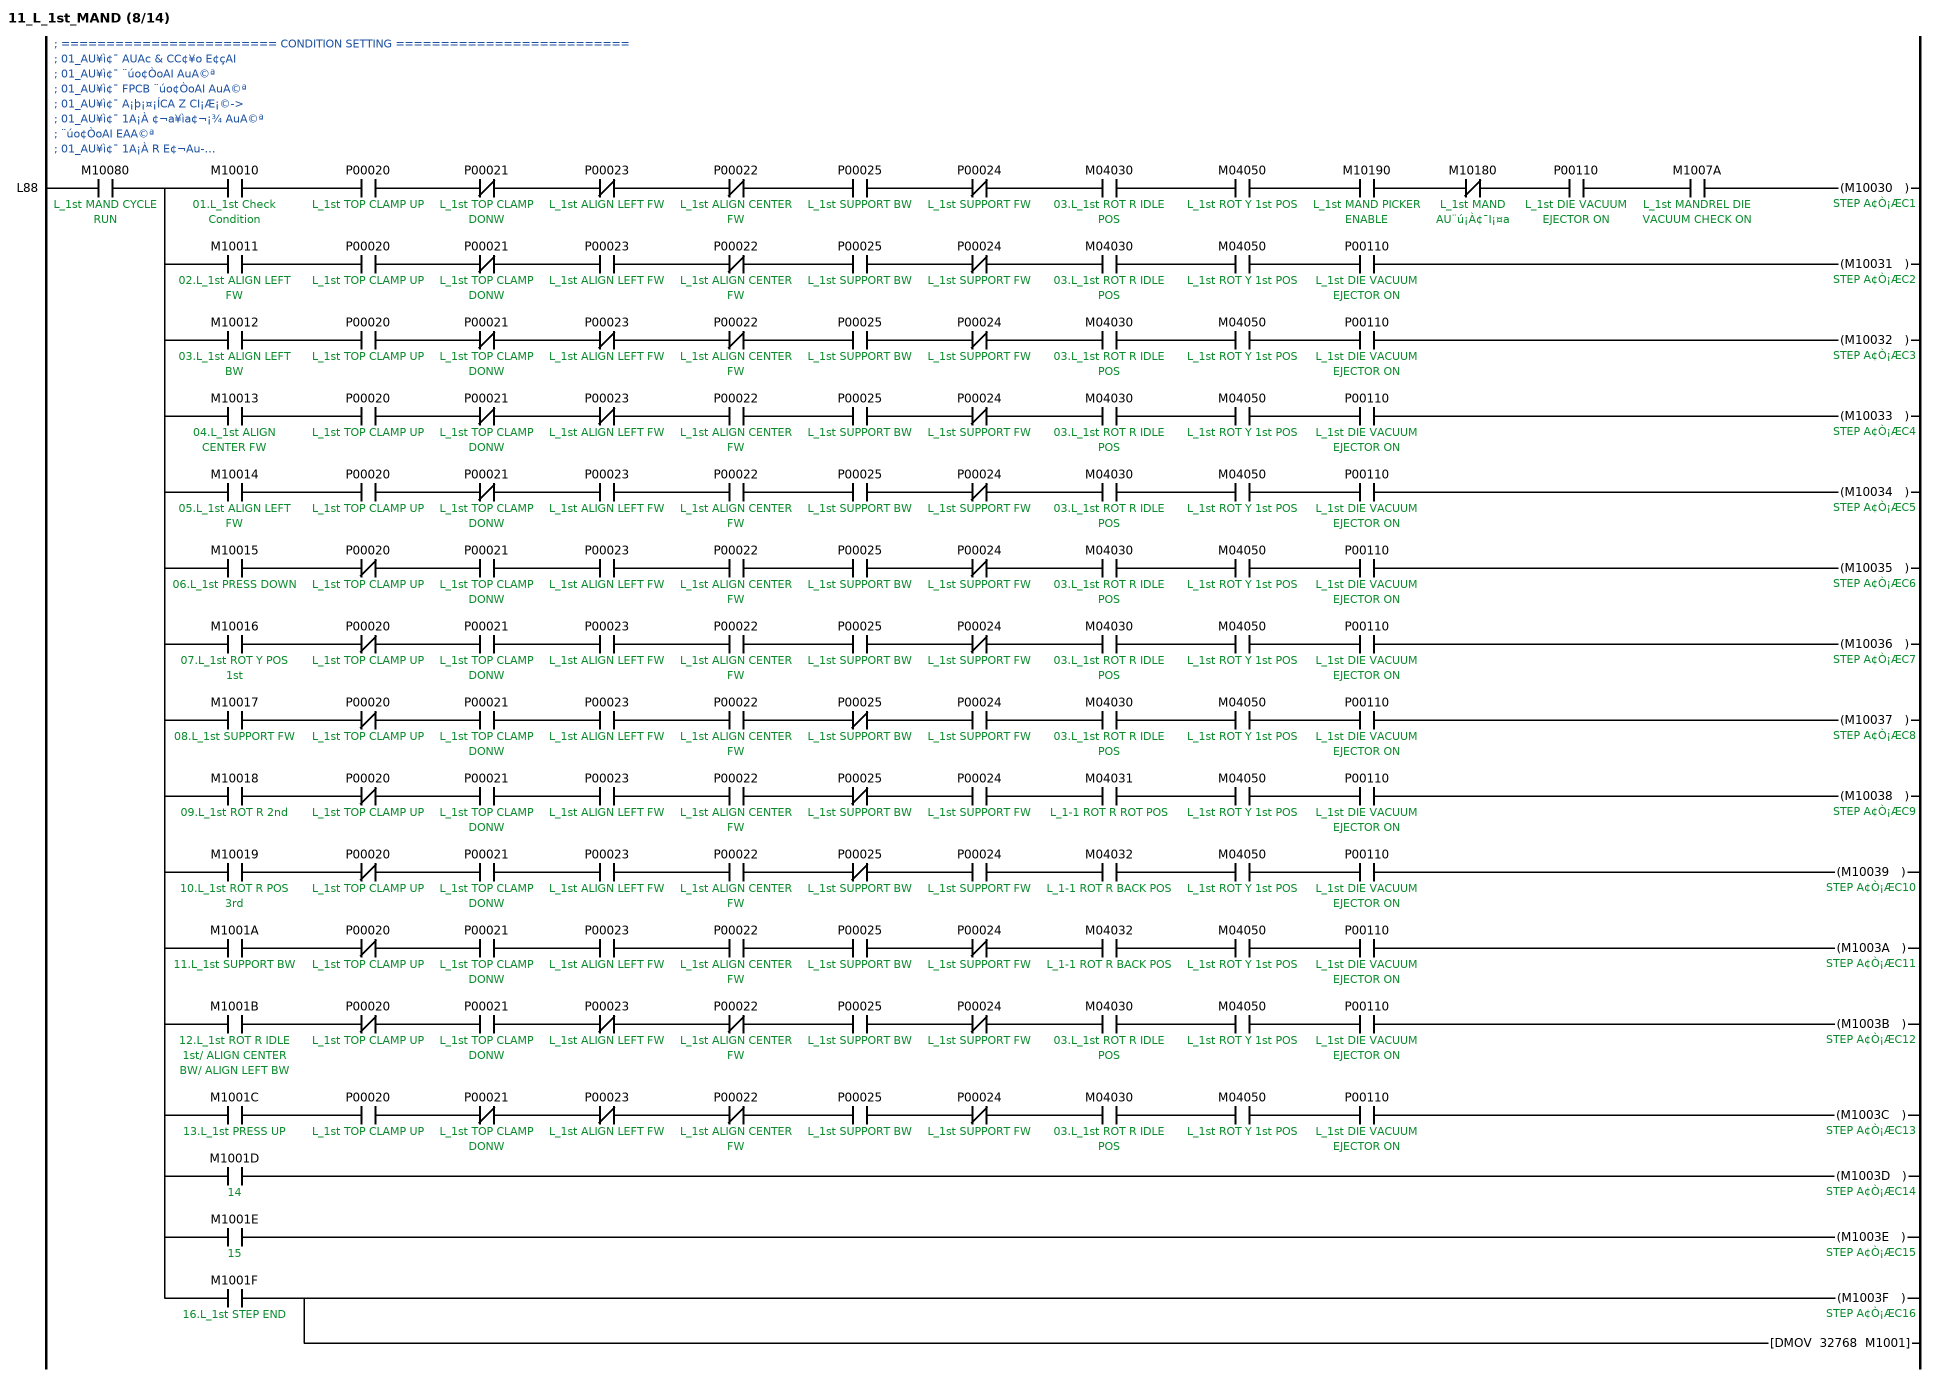
// ======================== CONDITION SETTING ==========================
; L88
LOAD      M10080	// L_1st MAND CYCLE RUN
MPUSH
AND       M10010	// 01.L_1st Check Condition
AND       P00020	// L_1st TOP CLAMP UP
AND NOT   P00021	// L_1st TOP CLAMP DONW
AND NOT   P00023	// L_1st ALIGN LEFT FW
AND NOT   P00022	// L_1st ALIGN CENTER FW
AND       P00025	// L_1st SUPPORT BW
AND NOT   P00024	// L_1st SUPPORT FW
AND       M04030	// 03.L_1st ROT R IDLE POS
AND       M04050	// L_1st ROT Y 1st POS
AND       M10190	// L_1st MAND PICKER ENABLE
AND NOT   M10180	// L_1st MAND AU¨ú¡À¢¯I¡¤a
AND       P00110	// L_1st DIE VACUUM EJECTOR ON
AND       M1007A	// L_1st MANDREL DIE VACUUM CHECK ON
OUT       M10030	// STEP A¢Ò¡ÆC1
MLOAD
AND       M10011	// 02.L_1st ALIGN LEFT FW
AND       P00020	// L_1st TOP CLAMP UP
AND NOT   P00021	// L_1st TOP CLAMP DONW
AND       P00023	// L_1st ALIGN LEFT FW
AND NOT   P00022	// L_1st ALIGN CENTER FW
AND       P00025	// L_1st SUPPORT BW
AND NOT   P00024	// L_1st SUPPORT FW
AND       M04030	// 03.L_1st ROT R IDLE POS
AND       M04050	// L_1st ROT Y 1st POS
AND       P00110	// L_1st DIE VACUUM EJECTOR ON
OUT       M10031	// STEP A¢Ò¡ÆC2
MLOAD
AND       M10012	// 03.L_1st ALIGN LEFT BW
AND       P00020	// L_1st TOP CLAMP UP
AND NOT   P00021	// L_1st TOP CLAMP DONW
AND NOT   P00023	// L_1st ALIGN LEFT FW
AND NOT   P00022	// L_1st ALIGN CENTER FW
AND       P00025	// L_1st SUPPORT BW
AND NOT   P00024	// L_1st SUPPORT FW
AND       M04030	// 03.L_1st ROT R IDLE POS
AND       M04050	// L_1st ROT Y 1st POS
AND       P00110	// L_1st DIE VACUUM EJECTOR ON
OUT       M10032	// STEP A¢Ò¡ÆC3
MLOAD
AND       M10013	// 04.L_1st ALIGN CENTER FW
AND       P00020	// L_1st TOP CLAMP UP
AND NOT   P00021	// L_1st TOP CLAMP DONW
AND NOT   P00023	// L_1st ALIGN LEFT FW
AND       P00022	// L_1st ALIGN CENTER FW
AND       P00025	// L_1st SUPPORT BW
AND NOT   P00024	// L_1st SUPPORT FW
AND       M04030	// 03.L_1st ROT R IDLE POS
AND       M04050	// L_1st ROT Y 1st POS
AND       P00110	// L_1st DIE VACUUM EJECTOR ON
OUT       M10033	// STEP A¢Ò¡ÆC4
MLOAD
AND       M10014	// 05.L_1st ALIGN LEFT FW
AND       P00020	// L_1st TOP CLAMP UP
AND NOT   P00021	// L_1st TOP CLAMP DONW
AND       P00023	// L_1st ALIGN LEFT FW
AND       P00022	// L_1st ALIGN CENTER FW
AND       P00025	// L_1st SUPPORT BW
AND NOT   P00024	// L_1st SUPPORT FW
AND       M04030	// 03.L_1st ROT R IDLE POS
AND       M04050	// L_1st ROT Y 1st POS
AND       P00110	// L_1st DIE VACUUM EJECTOR ON
OUT       M10034	// STEP A¢Ò¡ÆC5
MLOAD
AND       M10015	// 06.L_1st PRESS DOWN
AND NOT   P00020	// L_1st TOP CLAMP UP
AND       P00021	// L_1st TOP CLAMP DONW
AND       P00023	// L_1st ALIGN LEFT FW
AND       P00022	// L_1st ALIGN CENTER FW
AND       P00025	// L_1st SUPPORT BW
AND NOT   P00024	// L_1st SUPPORT FW
AND       M04030	// 03.L_1st ROT R IDLE POS
AND       M04050	// L_1st ROT Y 1st POS
AND       P00110	// L_1st DIE VACUUM EJECTOR ON
OUT       M10035	// STEP A¢Ò¡ÆC6
MLOAD
AND       M10016	// 07.L_1st ROT Y POS 1st
AND NOT   P00020	// L_1st TOP CLAMP UP
AND       P00021	// L_1st TOP CLAMP DONW
AND       P00023	// L_1st ALIGN LEFT FW
AND       P00022	// L_1st ALIGN CENTER FW
AND       P00025	// L_1st SUPPORT BW
AND NOT   P00024	// L_1st SUPPORT FW
AND       M04030	// 03.L_1st ROT R IDLE POS
AND       M04050	// L_1st ROT Y 1st POS
AND       P00110	// L_1st DIE VACUUM EJECTOR ON
OUT       M10036	// STEP A¢Ò¡ÆC7
MLOAD
AND       M10017	// 08.L_1st SUPPORT FW
AND NOT   P00020	// L_1st TOP CLAMP UP
AND       P00021	// L_1st TOP CLAMP DONW
AND       P00023	// L_1st ALIGN LEFT FW
AND       P00022	// L_1st ALIGN CENTER FW
AND NOT   P00025	// L_1st SUPPORT BW
AND       P00024	// L_1st SUPPORT FW
AND       M04030	// 03.L_1st ROT R IDLE POS
AND       M04050	// L_1st ROT Y 1st POS
AND       P00110	// L_1st DIE VACUUM EJECTOR ON
OUT       M10037	// STEP A¢Ò¡ÆC8
MLOAD
AND       M10018	// 09.L_1st ROT R 2nd
AND NOT   P00020	// L_1st TOP CLAMP UP
AND       P00021	// L_1st TOP CLAMP DONW
AND       P00023	// L_1st ALIGN LEFT FW
AND       P00022	// L_1st ALIGN CENTER FW
AND NOT   P00025	// L_1st SUPPORT BW
AND       P00024	// L_1st SUPPORT FW
AND       M04031	// L_1-1 ROT R ROT POS
AND       M04050	// L_1st ROT Y 1st POS
AND       P00110	// L_1st DIE VACUUM EJECTOR ON
OUT       M10038	// STEP A¢Ò¡ÆC9
MLOAD
AND       M10019	// 10.L_1st ROT R POS 3rd
AND NOT   P00020	// L_1st TOP CLAMP UP
AND       P00021	// L_1st TOP CLAMP DONW
AND       P00023	// L_1st ALIGN LEFT FW
AND       P00022	// L_1st ALIGN CENTER FW
AND NOT   P00025	// L_1st SUPPORT BW
AND       P00024	// L_1st SUPPORT FW
AND       M04032	// L_1-1 ROT R BACK POS
AND       M04050	// L_1st ROT Y 1st POS
AND       P00110	// L_1st DIE VACUUM EJECTOR ON
OUT       M10039	// STEP A¢Ò¡ÆC10
MLOAD
AND       M1001A	// 11.L_1st SUPPORT BW
AND NOT   P00020	// L_1st TOP CLAMP UP
AND       P00021	// L_1st TOP CLAMP DONW
AND       P00023	// L_1st ALIGN LEFT FW
AND       P00022	// L_1st ALIGN CENTER FW
AND       P00025	// L_1st SUPPORT BW
AND NOT   P00024	// L_1st SUPPORT FW
AND       M04032	// L_1-1 ROT R BACK POS
AND       M04050	// L_1st ROT Y 1st POS
AND       P00110	// L_1st DIE VACUUM EJECTOR ON
OUT       M1003A	// STEP A¢Ò¡ÆC11
MLOAD
AND       M1001B	// 12.L_1st ROT R IDLE 1st/ ALIGN CENTER BW/ ALIGN LEFT BW
AND NOT   P00020	// L_1st TOP CLAMP UP
AND       P00021	// L_1st TOP CLAMP DONW
AND NOT   P00023	// L_1st ALIGN LEFT FW
AND NOT   P00022	// L_1st ALIGN CENTER FW
AND       P00025	// L_1st SUPPORT BW
AND NOT   P00024	// L_1st SUPPORT FW
AND       M04030	// 03.L_1st ROT R IDLE POS
AND       M04050	// L_1st ROT Y 1st POS
AND       P00110	// L_1st DIE VACUUM EJECTOR ON
OUT       M1003B	// STEP A¢Ò¡ÆC12
MLOAD
AND       M1001C	// 13.L_1st PRESS UP
AND       P00020	// L_1st TOP CLAMP UP
AND NOT   P00021	// L_1st TOP CLAMP DONW
AND NOT   P00023	// L_1st ALIGN LEFT FW
AND NOT   P00022	// L_1st ALIGN CENTER FW
AND       P00025	// L_1st SUPPORT BW
AND NOT   P00024	// L_1st SUPPORT FW
AND       M04030	// 03.L_1st ROT R IDLE POS
AND       M04050	// L_1st ROT Y 1st POS
AND       P00110	// L_1st DIE VACUUM EJECTOR ON
OUT       M1003C	// STEP A¢Ò¡ÆC13
MLOAD
AND       M1001D	// 14
OUT       M1003D	// STEP A¢Ò¡ÆC14
MLOAD
AND       M1001E	// 15
OUT       M1003E	// STEP A¢Ò¡ÆC15
MPOP
AND       M1001F	// 16.L_1st STEP END
OUT       M1003F	// STEP A¢Ò¡ÆC16
DMOV      32768 M1001
// output comment: 01_AU¥ì¢¯ AUAc & CC¢¥o E¢çAI
// output comment: 01_AU¥ì¢¯ ¨úo¢ÒoAI AuA©ª
// output comment: 01_AU¥ì¢¯ FPCB ¨úo¢ÒoAI AuA©ª
// output comment: 01_AU¥ì¢¯ A¡þ¡¤¡ÍCA Z CI¡Æ¡©->
// output comment: 01_AU¥ì¢¯ 1A¡À ¢¬a¥ìa¢¬¡¾ AuA©ª ¨úo¢ÒoAI EAA©ª
// output comment: 01_AU¥ì¢¯ 1A¡À R E¢¬Au->
// output comment: 01_AU¥ì¢¯ 1A¡À R ¨¬©ö¡¾I->
// output comment: 01_AU¥ì¢¯ 1A¡À ¢¬a¥ìa¢¬¡¾ EAA©ª
// output comment: 01_AU¥ì¢¯ R ¢¥e¡¾a -> ¡ío¨¬I ¡ío¨öA

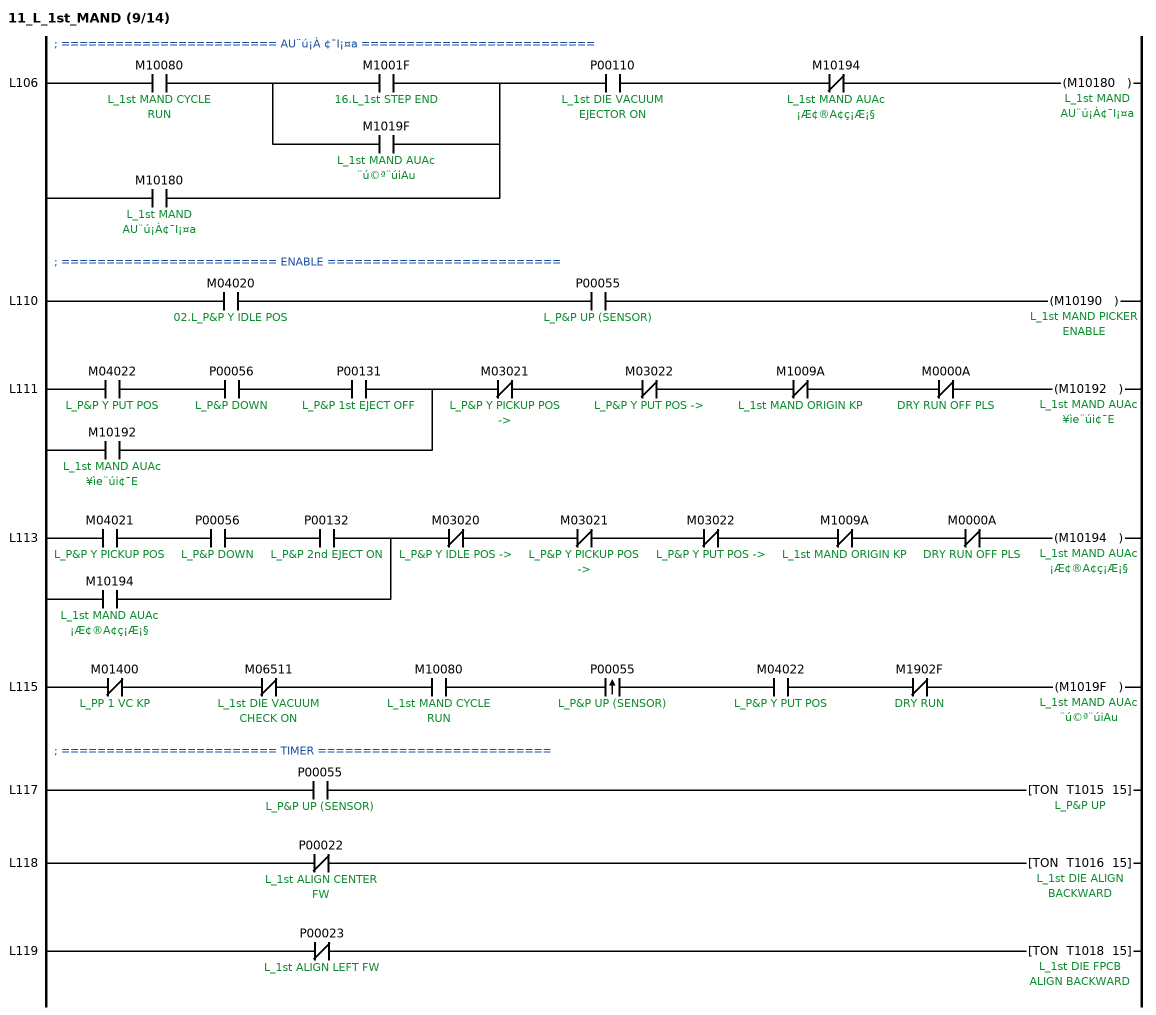
// ======================== AU¨ú¡À ¢¯I¡¤a ==========================
; L106
LOAD      M10080	// L_1st MAND CYCLE RUN
LOAD      M1001F	// 16.L_1st STEP END
OR        M1019F	// L_1st MAND AUAc ¨ú©ª¨úiAu
AND LOAD
OR        M10180	// L_1st MAND AU¨ú¡À¢¯I¡¤a
AND       P00110	// L_1st DIE VACUUM EJECTOR ON
AND NOT   M10194	// L_1st MAND AUAc ¡Æ¢®A¢ç¡Æ¡§
OUT       M10180	// L_1st MAND AU¨ú¡À¢¯I¡¤a
// ======================== ENABLE ==========================
; L110
LOAD      M04020	// 02.L_P&P Y IDLE POS
AND       P00055	// L_P&P UP (SENSOR)
OUT       M10190	// L_1st MAND PICKER ENABLE
; L111
LOAD      M04022	// L_P&P Y PUT POS
AND       P00056	// L_P&P DOWN
AND       P00131	// L_P&P 1st EJECT OFF
OR        M10192	// L_1st MAND AUAc ¥ìe¨úi¢¯E
AND NOT   M03021	// L_P&P Y PICKUP POS ->
AND NOT   M03022	// L_P&P Y PUT POS ->
AND NOT   M1009A	// L_1st MAND ORIGIN KP
AND NOT   M0000A	// DRY RUN OFF PLS
OUT       M10192	// L_1st MAND AUAc ¥ìe¨úi¢¯E
; L113
LOAD      M04021	// L_P&P Y PICKUP POS
AND       P00056	// L_P&P DOWN
AND       P00132	// L_P&P 2nd EJECT ON
OR        M10194	// L_1st MAND AUAc ¡Æ¢®A¢ç¡Æ¡§
AND NOT   M03020	// L_P&P Y IDLE POS ->
AND NOT   M03021	// L_P&P Y PICKUP POS ->
AND NOT   M03022	// L_P&P Y PUT POS ->
AND NOT   M1009A	// L_1st MAND ORIGIN KP
AND NOT   M0000A	// DRY RUN OFF PLS
OUT       M10194	// L_1st MAND AUAc ¡Æ¢®A¢ç¡Æ¡§
; L115
LOAD NOT  M01400	// L_PP 1 VC KP
AND NOT   M06511	// L_1st DIE VACUUM CHECK ON
AND       M10080	// L_1st MAND CYCLE RUN
ANDP      P00055	// L_P&P UP (SENSOR)
AND       M04022	// L_P&P Y PUT POS
AND NOT   M1902F	// DRY RUN
OUT       M1019F	// L_1st MAND AUAc ¨ú©ª¨úiAu
// ======================== TIMER ==========================
; L117
LOAD      P00055	// L_P&P UP (SENSOR)
TON       T1015 15	// L_P&P UP
; L118
LOAD NOT  P00022	// L_1st ALIGN CENTER FW
TON       T1016 15	// L_1st DIE ALIGN BACKWARD
; L119
LOAD NOT  P00023	// L_1st ALIGN LEFT FW
TON       T1018 15	// L_1st DIE FPCB ALIGN BACKWARD

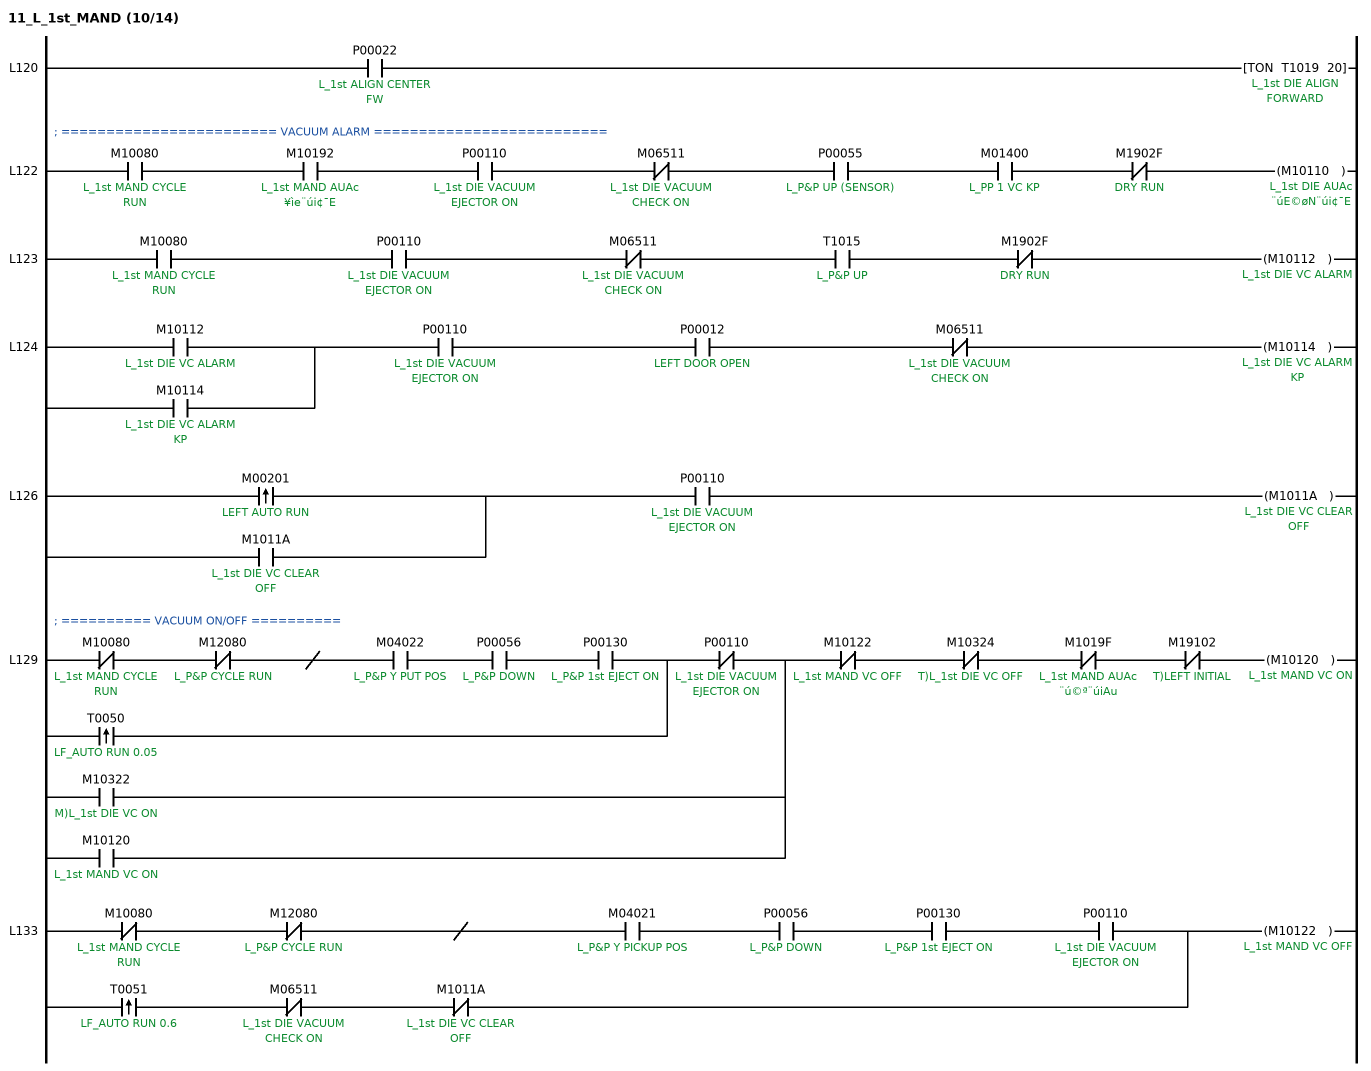
; L120
LOAD      P00022	// L_1st ALIGN CENTER FW
TON       T1019 20	// L_1st DIE ALIGN FORWARD
// ======================== VACUUM ALARM ==========================
; L122
LOAD      M10080	// L_1st MAND CYCLE RUN
AND       M10192	// L_1st MAND AUAc ¥ìe¨úi¢¯E
AND       P00110	// L_1st DIE VACUUM EJECTOR ON
AND NOT   M06511	// L_1st DIE VACUUM CHECK ON
AND       P00055	// L_P&P UP (SENSOR)
AND       M01400	// L_PP 1 VC KP
AND NOT   M1902F	// DRY RUN
OUT       M10110	// L_1st DIE AUAc ¨úE©øN¨úi¢¯E
; L123
LOAD      M10080	// L_1st MAND CYCLE RUN
AND       P00110	// L_1st DIE VACUUM EJECTOR ON
AND NOT   M06511	// L_1st DIE VACUUM CHECK ON
AND       T1015	// L_P&P UP
AND NOT   M1902F	// DRY RUN
OUT       M10112	// L_1st DIE VC ALARM
; L124
LOAD      M10112	// L_1st DIE VC ALARM
OR        M10114	// L_1st DIE VC ALARM KP
AND       P00110	// L_1st DIE VACUUM EJECTOR ON
AND       P00012	// LEFT DOOR OPEN
AND NOT   M06511	// L_1st DIE VACUUM CHECK ON
OUT       M10114	// L_1st DIE VC ALARM KP
; L126
LOADP     M00201	// LEFT AUTO RUN
OR        M1011A	// L_1st DIE VC CLEAR OFF
AND       P00110	// L_1st DIE VACUUM EJECTOR ON
OUT       M1011A	// L_1st DIE VC CLEAR OFF
// ========== VACUUM ON/OFF ==========
; L129
LOAD NOT  M10080	// L_1st MAND CYCLE RUN
AND NOT   M12080	// L_P&P CYCLE RUN
NOT
AND       M04022	// L_P&P Y PUT POS
AND       P00056	// L_P&P DOWN
AND       P00130	// L_P&P 1st EJECT ON
ORP       T0050	// LF_AUTO RUN 0.05
AND NOT   P00110	// L_1st DIE VACUUM EJECTOR ON
OR        M10322	// M)L_1st DIE VC ON
OR        M10120	// L_1st MAND VC ON
AND NOT   M10122	// L_1st MAND VC OFF
AND NOT   M10324	// T)L_1st DIE VC OFF
AND NOT   M1019F	// L_1st MAND AUAc ¨ú©ª¨úiAu
AND NOT   M19102	// T)LEFT INITIAL
OUT       M10120	// L_1st MAND VC ON
; L133
LOAD NOT  M10080	// L_1st MAND CYCLE RUN
AND NOT   M12080	// L_P&P CYCLE RUN
NOT
AND       M04021	// L_P&P Y PICKUP POS
AND       P00056	// L_P&P DOWN
AND       P00130	// L_P&P 1st EJECT ON
AND       P00110	// L_1st DIE VACUUM EJECTOR ON
LOADP     T0051	// LF_AUTO RUN 0.6
AND NOT   M06511	// L_1st DIE VACUUM CHECK ON
AND NOT   M1011A	// L_1st DIE VC CLEAR OFF
OR LOAD
OUT       M10122	// L_1st MAND VC OFF

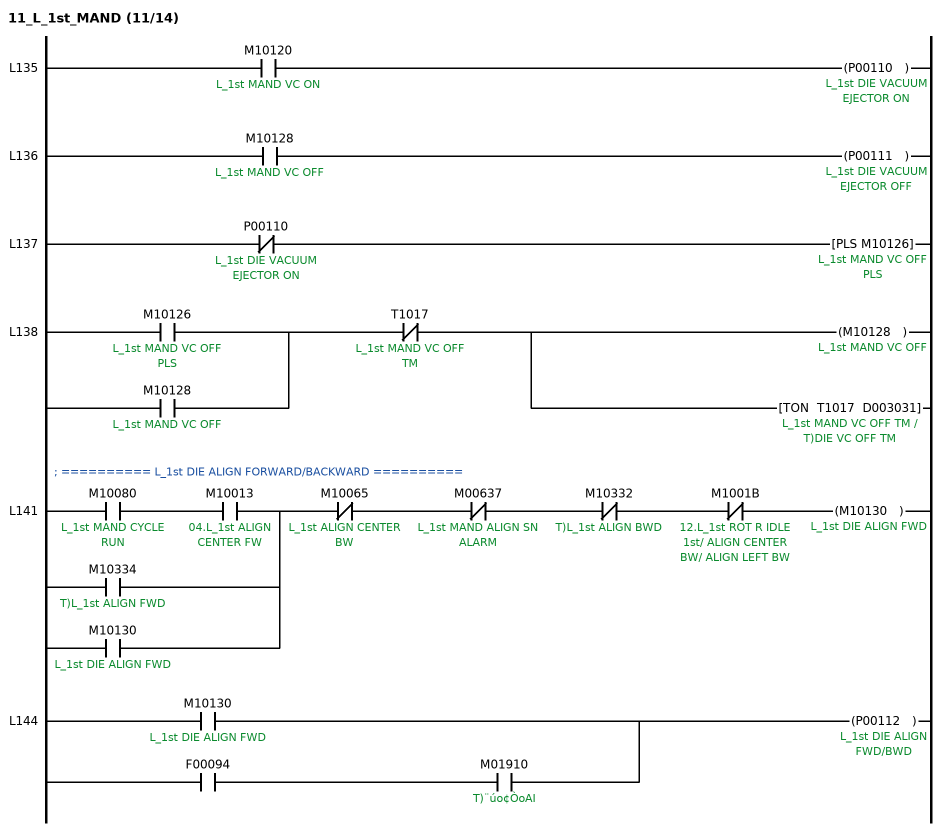
; L135
LOAD      M10120	// L_1st MAND VC ON
OUT       P00110	// L_1st DIE VACUUM EJECTOR ON
; L136
LOAD      M10128	// L_1st MAND VC OFF
OUT       P00111	// L_1st DIE VACUUM EJECTOR OFF
; L137
LOAD NOT  P00110	// L_1st DIE VACUUM EJECTOR ON
OUTP      M10126	// L_1st MAND VC OFF PLS
; L138
LOAD      M10126	// L_1st MAND VC OFF PLS
OR        M10128	// L_1st MAND VC OFF
AND NOT   T1017	// L_1st MAND VC OFF TM
OUT       M10128	// L_1st MAND VC OFF
TON       T1017 D003031	// L_1st MAND VC OFF TM / T)DIE VC OFF TM
// ========== L_1st DIE ALIGN FORWARD/BACKWARD ==========
; L141
LOAD      M10080	// L_1st MAND CYCLE RUN
AND       M10013	// 04.L_1st ALIGN CENTER FW
OR        M10334	// T)L_1st ALIGN FWD
OR        M10130	// L_1st DIE ALIGN FWD
AND NOT   M10065	// L_1st ALIGN CENTER BW
AND NOT   M00637	// L_1st MAND ALIGN SN ALARM
AND NOT   M10332	// T)L_1st ALIGN BWD
AND NOT   M1001B	// 12.L_1st ROT R IDLE 1st/ ALIGN CENTER BW/ ALIGN LEFT BW
OUT       M10130	// L_1st DIE ALIGN FWD
; L144
LOAD      M10130	// L_1st DIE ALIGN FWD
LOAD      F00094
AND       M01910	// T)¨úo¢ÒoAI
OR LOAD
OUT       P00112	// L_1st DIE ALIGN FWD/BWD

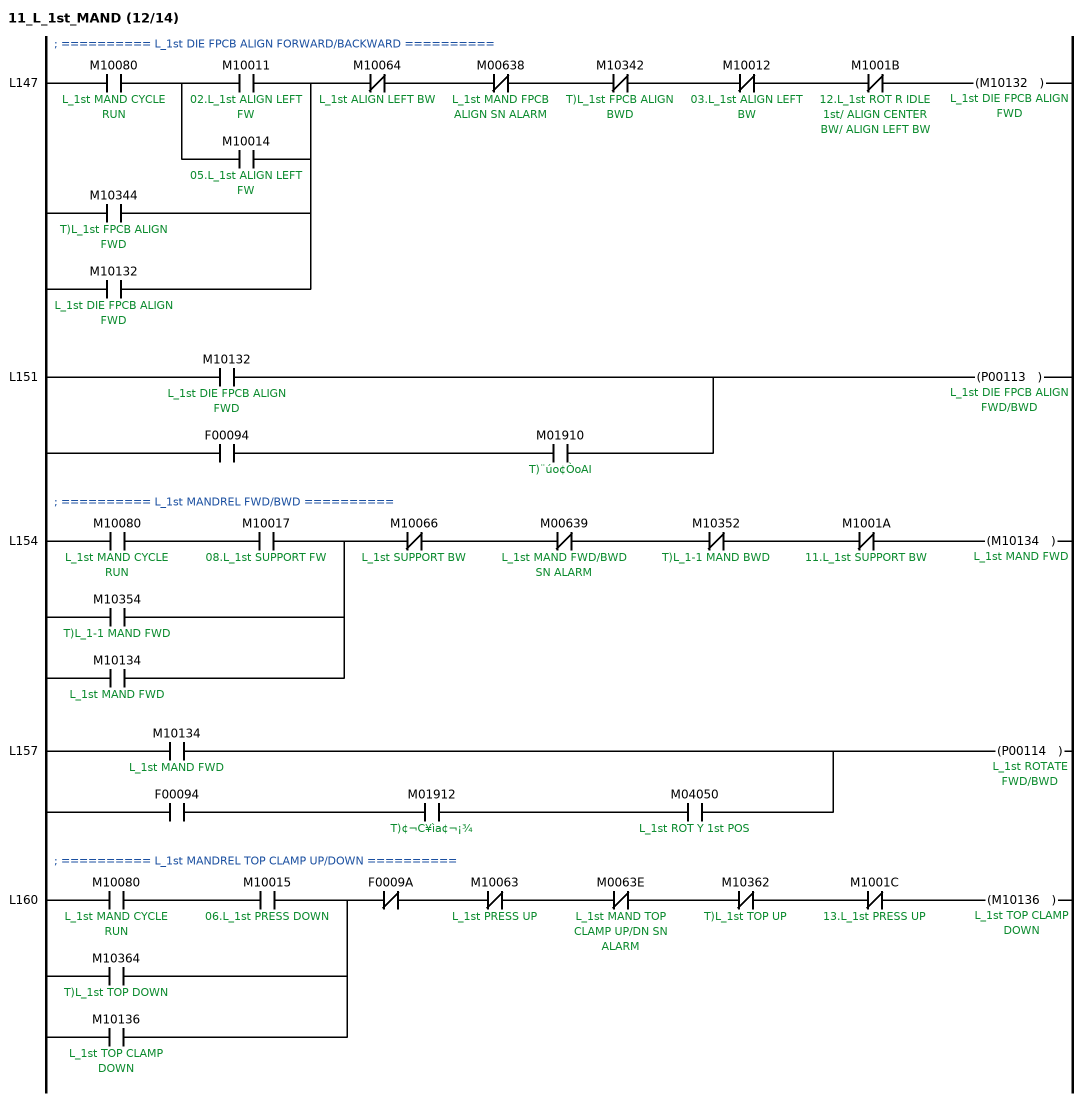
// ========== L_1st DIE FPCB ALIGN FORWARD/BACKWARD ==========
; L147
LOAD      M10080	// L_1st MAND CYCLE RUN
LOAD      M10011	// 02.L_1st ALIGN LEFT FW
OR        M10014	// 05.L_1st ALIGN LEFT FW
AND LOAD
OR        M10344	// T)L_1st FPCB ALIGN FWD
OR        M10132	// L_1st DIE FPCB ALIGN FWD
AND NOT   M10064	// L_1st ALIGN LEFT BW
AND NOT   M00638	// L_1st MAND FPCB ALIGN SN ALARM
AND NOT   M10342	// T)L_1st FPCB ALIGN BWD
AND NOT   M10012	// 03.L_1st ALIGN LEFT BW
AND NOT   M1001B	// 12.L_1st ROT R IDLE 1st/ ALIGN CENTER BW/ ALIGN LEFT BW
OUT       M10132	// L_1st DIE FPCB ALIGN FWD
; L151
LOAD      M10132	// L_1st DIE FPCB ALIGN FWD
LOAD      F00094
AND       M01910	// T)¨úo¢ÒoAI
OR LOAD
OUT       P00113	// L_1st DIE FPCB ALIGN FWD/BWD
// ========== L_1st MANDREL FWD/BWD ==========
; L154
LOAD      M10080	// L_1st MAND CYCLE RUN
AND       M10017	// 08.L_1st SUPPORT FW
OR        M10354	// T)L_1-1 MAND FWD
OR        M10134	// L_1st MAND FWD
AND NOT   M10066	// L_1st SUPPORT BW
AND NOT   M00639	// L_1st MAND FWD/BWD SN ALARM
AND NOT   M10352	// T)L_1-1 MAND BWD
AND NOT   M1001A	// 11.L_1st SUPPORT BW
OUT       M10134	// L_1st MAND FWD
; L157
LOAD      M10134	// L_1st MAND FWD
LOAD      F00094
AND       M01912	// T)¢¬C¥ìa¢¬¡¾
AND       M04050	// L_1st ROT Y 1st POS
OR LOAD
OUT       P00114	// L_1st ROTATE FWD/BWD
// ========== L_1st MANDREL TOP CLAMP UP/DOWN ==========
; L160
LOAD      M10080	// L_1st MAND CYCLE RUN
AND       M10015	// 06.L_1st PRESS DOWN
OR        M10364	// T)L_1st TOP DOWN
OR        M10136	// L_1st TOP CLAMP DOWN
AND NOT   F0009A
AND NOT   M10063	// L_1st PRESS UP
AND NOT   M0063E	// L_1st MAND TOP CLAMP UP/DN SN ALARM
AND NOT   M10362	// T)L_1st TOP UP
AND NOT   M1001C	// 13.L_1st PRESS UP
OUT       M10136	// L_1st TOP CLAMP DOWN

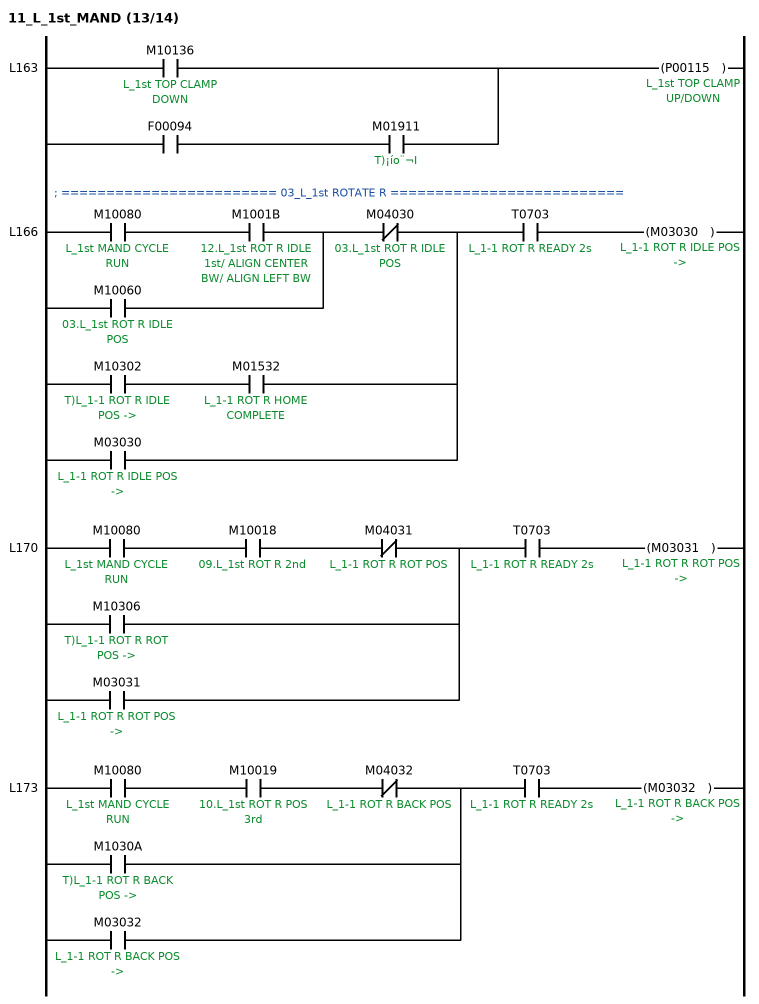
; L163
LOAD      M10136	// L_1st TOP CLAMP DOWN
LOAD      F00094
AND       M01911	// T)¡ío¨¬I
OR LOAD
OUT       P00115	// L_1st TOP CLAMP UP/DOWN
// ======================== 03_L_1st ROTATE R ==========================
; L166
LOAD      M10080	// L_1st MAND CYCLE RUN
AND       M1001B	// 12.L_1st ROT R IDLE 1st/ ALIGN CENTER BW/ ALIGN LEFT BW
OR        M10060	// 03.L_1st ROT R IDLE POS
AND NOT   M04030	// 03.L_1st ROT R IDLE POS
LOAD      M10302	// T)L_1-1 ROT R IDLE POS ->
AND       M01532	// L_1-1 ROT R HOME COMPLETE
OR LOAD
OR        M03030	// L_1-1 ROT R IDLE POS ->
AND       T0703	// L_1-1 ROT R READY 2s
OUT       M03030	// L_1-1 ROT R IDLE POS ->
; L170
LOAD      M10080	// L_1st MAND CYCLE RUN
AND       M10018	// 09.L_1st ROT R 2nd
AND NOT   M04031	// L_1-1 ROT R ROT POS
OR        M10306	// T)L_1-1 ROT R ROT POS ->
OR        M03031	// L_1-1 ROT R ROT POS ->
AND       T0703	// L_1-1 ROT R READY 2s
OUT       M03031	// L_1-1 ROT R ROT POS ->
; L173
LOAD      M10080	// L_1st MAND CYCLE RUN
AND       M10019	// 10.L_1st ROT R POS 3rd
AND NOT   M04032	// L_1-1 ROT R BACK POS
OR        M1030A	// T)L_1-1 ROT R BACK POS ->
OR        M03032	// L_1-1 ROT R BACK POS ->
AND       T0703	// L_1-1 ROT R READY 2s
OUT       M03032	// L_1-1 ROT R BACK POS ->

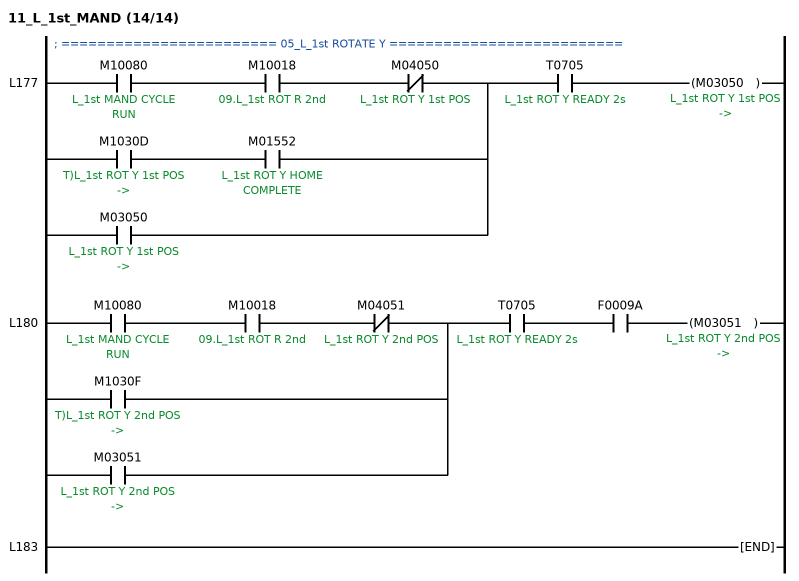
// ======================== 05_L_1st ROTATE Y ==========================
; L177
LOAD      M10080	// L_1st MAND CYCLE RUN
AND       M10018	// 09.L_1st ROT R 2nd
AND NOT   M04050	// L_1st ROT Y 1st POS
LOAD      M1030D	// T)L_1st ROT Y 1st POS ->
AND       M01552	// L_1st ROT Y HOME COMPLETE
OR LOAD
OR        M03050	// L_1st ROT Y 1st POS ->
AND       T0705	// L_1st ROT Y READY 2s
OUT       M03050	// L_1st ROT Y 1st POS ->
; L180
LOAD      M10080	// L_1st MAND CYCLE RUN
AND       M10018	// 09.L_1st ROT R 2nd
AND NOT   M04051	// L_1st ROT Y 2nd POS
OR        M1030F	// T)L_1st ROT Y 2nd POS ->
OR        M03051	// L_1st ROT Y 2nd POS ->
AND       T0705	// L_1st ROT Y READY 2s
AND       F0009A
OUT       M03051	// L_1st ROT Y 2nd POS ->
; L183
END

PROGRAM 12_L_2nd_MAND (task: ¨ö¨¬A¥ì CA¡¤I¡¾¡¿¡¤¡Í)

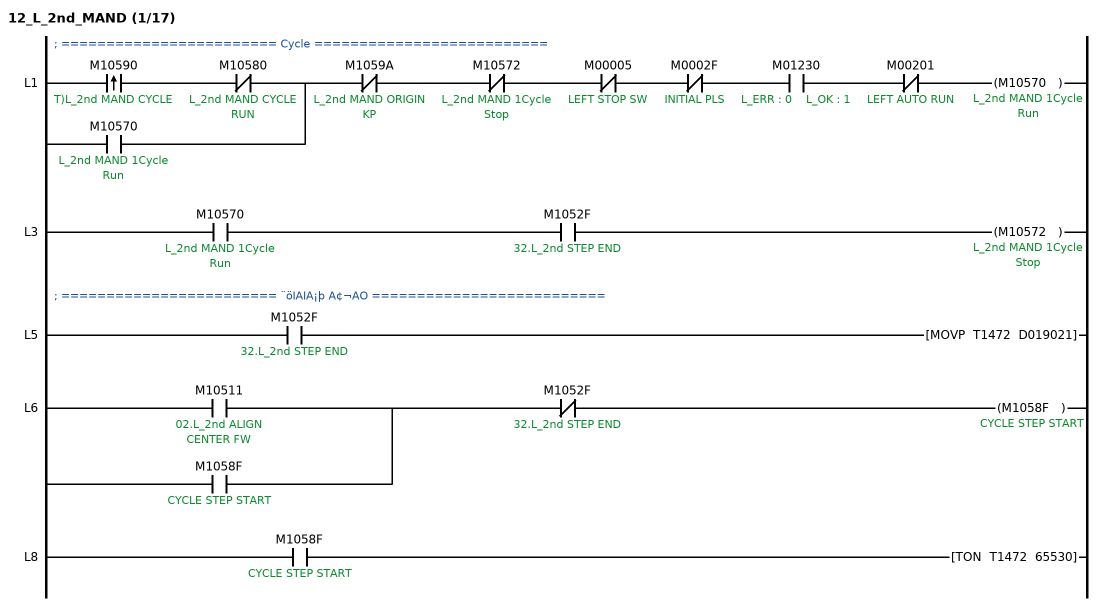
// ======================== Cycle ==========================
; L1
LOADP     M10590	// T)L_2nd MAND CYCLE
AND NOT   M10580	// L_2nd MAND CYCLE RUN
OR        M10570	// L_2nd MAND 1Cycle Run
AND NOT   M1059A	// L_2nd MAND ORIGIN KP
AND NOT   M10572	// L_2nd MAND 1Cycle Stop
AND NOT   M00005	// LEFT STOP SW
AND NOT   M0002F	// INITIAL PLS
AND       M01230	// L_ERR : 0    L_OK : 1
AND NOT   M00201	// LEFT AUTO RUN
OUT       M10570	// L_2nd MAND 1Cycle Run
; L3
LOAD      M10570	// L_2nd MAND 1Cycle Run
AND       M1052F	// 32.L_2nd STEP END
OUT       M10572	// L_2nd MAND 1Cycle Stop
// ======================== ¨öIAIA¡þ A¢¬AO ==========================
; L5
LOAD      M1052F	// 32.L_2nd STEP END
MOVP      T1472 D019021
; L6
LOAD      M10511	// 02.L_2nd ALIGN CENTER FW
OR        M1058F	// CYCLE STEP START
AND NOT   M1052F	// 32.L_2nd STEP END
OUT       M1058F	// CYCLE STEP START
; L8
LOAD      M1058F	// CYCLE STEP START
TON       T1472 65530

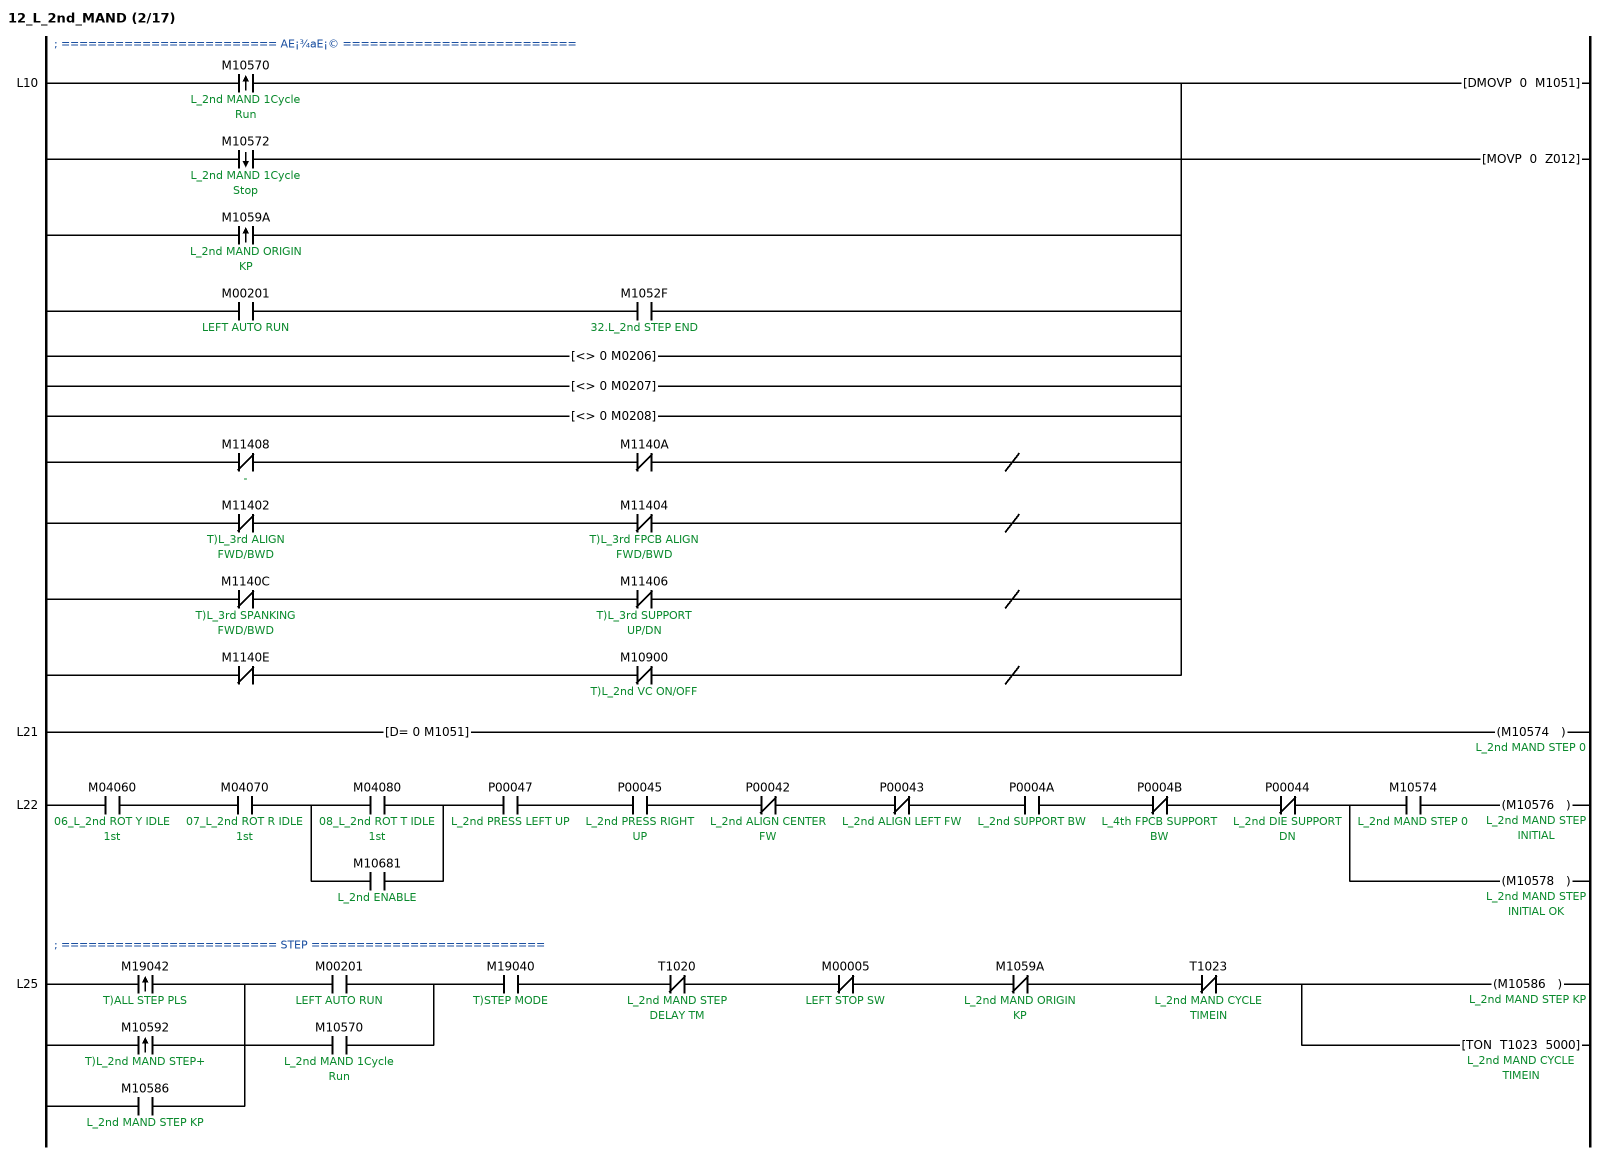
// ======================== AE¡¾aE¡© ==========================
; L10
LOADP     M10570	// L_2nd MAND 1Cycle Run
ORN       M10572	// L_2nd MAND 1Cycle Stop
ORP       M1059A	// L_2nd MAND ORIGIN KP
LOAD      M00201	// LEFT AUTO RUN
AND       M1052F	// 32.L_2nd STEP END
OR LOAD
OR<>      0 M0206
OR<>      0 M0207
OR<>      0 M0208
LOAD NOT  M11408	// -
AND NOT   M1140A
NOT
OR LOAD
LOAD NOT  M11402	// T)L_3rd ALIGN FWD/BWD
AND NOT   M11404	// T)L_3rd FPCB ALIGN FWD/BWD
NOT
OR LOAD
LOAD NOT  M1140C	// T)L_3rd SPANKING FWD/BWD
AND NOT   M11406	// T)L_3rd SUPPORT UP/DN
NOT
OR LOAD
LOAD NOT  M1140E
AND NOT   M10900	// T)L_2nd VC ON/OFF
NOT
OR LOAD
DMOVP     0 M1051
MOVP      0 Z012
; L21
LOADD=    0 M1051
OUT       M10574	// L_2nd MAND STEP 0
; L22
LOAD      M04060	// 06_L_2nd ROT Y IDLE 1st
AND       M04070	// 07_L_2nd ROT R IDLE 1st
LOAD      M04080	// 08_L_2nd ROT T IDLE 1st
OR        M10681	// L_2nd ENABLE
AND LOAD
AND       P00047	// L_2nd PRESS LEFT UP
AND       P00045	// L_2nd PRESS RIGHT UP
AND NOT   P00042	// L_2nd ALIGN CENTER FW
AND NOT   P00043	// L_2nd ALIGN LEFT FW
AND       P0004A	// L_2nd SUPPORT BW
AND NOT   P0004B	// L_4th FPCB SUPPORT BW
AND NOT   P00044	// L_2nd DIE SUPPORT DN
MPUSH
AND       M10574	// L_2nd MAND STEP 0
OUT       M10576	// L_2nd MAND STEP INITIAL
MPOP
OUT       M10578	// L_2nd MAND STEP INITIAL OK
// ======================== STEP ==========================
; L25
LOADP     M19042	// T)ALL STEP PLS
ORP       M10592	// T)L_2nd MAND STEP+
OR        M10586	// L_2nd MAND STEP KP
LOAD      M00201	// LEFT AUTO RUN
OR        M10570	// L_2nd MAND 1Cycle Run
AND LOAD
AND       M19040	// T)STEP MODE
AND NOT   T1020	// L_2nd MAND STEP DELAY TM
AND NOT   M00005	// LEFT STOP SW
AND NOT   M1059A	// L_2nd MAND ORIGIN KP
AND NOT   T1023	// L_2nd MAND CYCLE TIMEIN
OUT       M10586	// L_2nd MAND STEP KP
TON       T1023 5000	// L_2nd MAND CYCLE TIMEIN

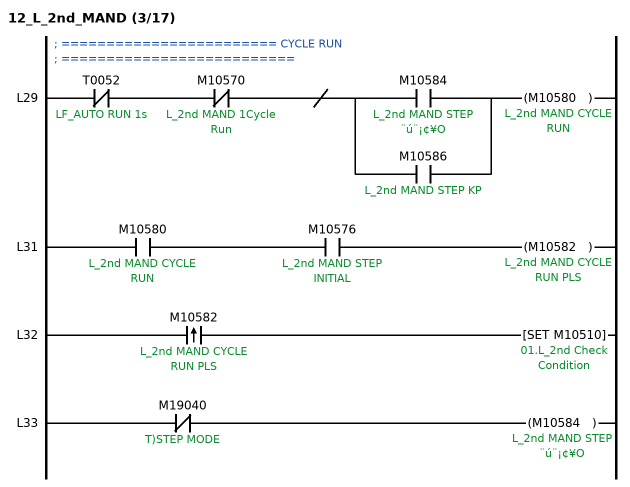
// ======================== CYCLE RUN ==========================
; L29
LOAD NOT  T0052	// LF_AUTO RUN 1s
AND NOT   M10570	// L_2nd MAND 1Cycle Run
NOT
LOAD      M10584	// L_2nd MAND STEP ¨ú¨¡¢¥O
OR        M10586	// L_2nd MAND STEP KP
AND LOAD
OUT       M10580	// L_2nd MAND CYCLE RUN
; L31
LOAD      M10580	// L_2nd MAND CYCLE RUN
AND       M10576	// L_2nd MAND STEP INITIAL
OUT       M10582	// L_2nd MAND CYCLE RUN PLS
; L32
LOADP     M10582	// L_2nd MAND CYCLE RUN PLS
SET       M10510	// 01.L_2nd Check Condition
; L33
LOAD NOT  M19040	// T)STEP MODE
OUT       M10584	// L_2nd MAND STEP ¨ú¨¡¢¥O

